// SIMATIC STEP 7 (V5.x) project EuroAsiaFood_V00_00_01
// station: Hardware
// station: SIMATIC 300(1)
// station: P_ADR_BUS
// station: Hardware
// station: SIMATIC 300(1)
// station: P_ADR_BUS

SYMBOL_TABLE
"CMs_SIMULATION_DB"	DB 2	FB 2	// Simulation
"DB3 CPU Daten"	DB 3	DB 3	// Globaldaten
"DB4 Motordaten für FUs"	DB 4	DB 4	// Motordaten für Frequenzumformer
"DB30 Daten von/an FG"	DB 30	FB 30
"DB32 Inputs"	DB 32	FB 32
"DB33 Outputs"	DB 33	FB 33
"DB34 Faults"	DB 34	FB 34
"DB35 Acknolegments"	DB 35	DB 35	// Quittierungen
"DB92 Eingänge AVP"	DB 92	FB 92
"CMs_MOTOR_1Q1I_DB"	DB 901	FB 901	// Motor 1QII
"LINE1"	DB 1000	FB 1000	// Line FB
"CONTAINERSTATION CST01"	DB 1001	FB 1001
"RECEIVER REC01"	DB 1011	FB 1011
"REC01"	DB 1012	FB 1011
"VP01"	DB 1051	FB 1051
"VACUUM PUMP VP01_02 SF01"	DB 1081	FB 1081
"RecipeData"	DB 1111	DB 1111	// Recipes
"test"	DB 2222	DB 2222
"FREQUENCY CONVERTERS"	DB 4900	FB 4900
"FC VACUUM PUMP"	DB 10001	FB 4901	// Vacuum Pump FC
"FC ROTARY FEEDER REC01"	DB 10002	FB 4901	// Rotary Feeder REC01 FC
"CMs_SIMULATION"	FB 2	FB 2	// Simulation
"FB4 Frequenzumformer"	FB 4	FB 4	// Frequenzumformer
"FB30 Daten von/an  FG"	FB 30	FB 30	// Daten von / an Farbgrafik
"FB31 Mode Objekte an FG"	FB 31	FB 31	// Mode der Objekte an Farbgrafik
"FB32 Eingaege an FG"	FB 32	FB 32	// Eingänge der an Farbgrafik
"FB33 Ausgaege an FG"	FB 33	FB 33	// Ausgänge der an Farbgrafik
"FB34 Störbearbeitung"	FB 34	FB 34	// Faults
"FB92 Eingänge AVP"	FB 92	FB 92	// reserve
"CMs_MOTOR_1Q1I"	FB 901	FB 901	// Motor 1QII
"****PRODUCTION****"	FB 1000	FB 1000	// Call Line FBs
"CONTAINERSTATION"	FB 1001	FB 1001	// HP01 and HP02
"RECEIVER"	FB 1011	FB 1011	// Receiver REC01
"VACUUM PUMP"	FB 1051	FB 1051
"VACUUMPUMP"	FB 1081	FB 1081	// BLOWER FB
"*** FCs ***"	FB 4900	FB 4900	// Frequency Converters
"FREQ.CONVERTER"	FB 4901	FB 4901	// Frequency Convertors Calls
"FU SEW DFE32B - PN_REL"	FB 6119	FB 6119
"FU SEW DFE32B - PN"	FB 60119	FB 60119	// SEW Profinet
"FC2 Taktgeber_Timernachb"	FC 2	FC 2	// Taktgeber mit Timernachbildung
"FC3 Timernachbildung"	FC 3	FC 3	// Timernachbildung SA,SE,SV,SI
"FC4 Blocktransfer ANY-Q"	FC 4	FC 4	// Block transferieren mit ANY-Zeiger als Quelle
"FC5 Blocktransfer"	FC 5	FC 5	// Block transferieren, Datenwort schreiben
"FC6 Datenbit zuw./abfr."	FC 6	FC 6	// Datenbit zuweisen oder abfragen
"FC7 Tabelle auslesen"	FC 7	FC 7	// Tabelle auslesen
"FC8 ANY-Zeiger zerlegen"	FC 8	FC 8	// ANY-Zeiger in DB,DW,Länge zerlegen
"FC10 Analogwert r/w"	FC 10	FC 10	// Analogwert lesen/schreiben
"FC13 Standardsignale"	FC 13	FC 13	// Standardsignale
"FC16 Störauswertung"	FC 16	FC 16	// Störauswertung
"FC20 Motor 1A1E"	FC 20	FC 20	// Motor Objekt 1 (1 Ausgang, 1 Eingang)
"FC21 Ventil 1A0-2E"	FC 21	FC 21	// Ventil Objekt 1 (1 Ausgang, 0-2 Eingänge)
"FC22 Ventil 2A2E"	FC 22	FC 22	// Ventil Objekt 2 (2 Ausgänge, 2Eingänge)
"FC23 Ventil 1-10A"	FC 23	FC 23	// Ventil Objekt 3 (Ansteuerung von max. 10 getakteten Ventilen)
"FC24 Binär-E"	FC 24	FC 24	// Binär-Eingangs Objekt
"FC25 Lamp"	FC 25	FC 25
"AnalogueIn"	FC 28	FC 28
"PressureAi"	FC 29	FC 29	// FU Objekt
"FC30 DB vorbelegen"	FC 30	FC 30	// Datenbaustein vorbelegen
"FC40 copy Obj-SST Master"	FC 40	FC 40	// Objekt-Schnittstelle kopieren Master
"FC41 copy Obj-SST Slave"	FC 41	FC 41	// Objekt-Schnittstelle kopieren Slave
"FC47 Tabelle schreiben"	FC 47	FC 47	// Eintrag in Tabelle schreiben
"FC104 Blocktransf. ANY-Z"	FC 104	FC 104
"FC113 Standardsignale 2"	FC 113	FC 113	// Standardsignale
"FC6079 SimAnalog"	FC 6079	FC 6079	// simulate analog signal using sin()
"FC6091 SimValve3A3E"	FC 6091	FC 6091	// simulate valve 3A3E (sealed hose diverter)
"FC6092 SimValveDOS"	FC 6092	FC 6092	// simulate valve 2A2E (dosing valve)
"FC6093 SimValveDS"	FC 6093	FC 6093	// simulate valve 2A2E (double seat)
"FC6094 SimMotor2A2E"	FC 6094	FC 6094	// simulate motor 2A2E
"FC6095 SimValve2A2E"	FC 6095	FC 6095	// simulate valve 2A2E
"FC6096 SimValve1AE1"	FC 6096	FC 6096	// simulate valve 1AE1
"FC6097 SimValve1A1E"	FC 6097	FC 6097	// simulate valve 1A1E
"FC6098 SimValve1A2E"	FC 6098	FC 6098	// simulate valve 1A2E
"FC6099 SimMotor1A1E"	FC 6099	FC 6099	// simulate motor 1A1E
"I 4.0"	I 4.0	BOOL
"02_01_101_Gn"	I 4.1	BOOL	// Production area PMP01 valve fresh air valve
"I 4.2"	I 4.2	BOOL
"02_02_101_Gp"	I 4.3	BOOL	// Production area REC01 valve angle valve
"I 4.4"	I 4.4	BOOL
"I 4.5"	I 4.5	BOOL
"I 4.6"	I 4.6	BOOL
"01_01_101_Gp"	I 4.7	BOOL	// Material preparation CST01 valve fresh air valve
"I 5.0"	I 5.0	BOOL
"02_01_101_Gp"	I 5.1	BOOL	// Production area PMP01 valve fresh air valve
"I 5.2"	I 5.2	BOOL
"02_02_101_Gn"	I 5.3	BOOL	// Production area REC01 valve angle valve
"I 5.4"	I 5.4	BOOL
"I 5.5"	I 5.5	BOOL
"I 5.6"	I 5.6	BOOL
"01_01_101_Gn"	I 5.7	BOOL	// Material preparation CST01 valve fresh air valve
"02_02_601_Lp"	I 6.0	BOOL	// Production area REC01 input high level indicator
"02_02_602_Gn"	I 6.1	BOOL	// Production area REC01 input pendulum flap
"I 6.2"	I 6.2	BOOL
"I 6.3"	I 6.3	BOOL
"I 6.4"	I 6.4	BOOL
"I 6.5"	I 6.5	BOOL
"I 6.6"	I 6.6	BOOL
"10_01_601_ES"	I 6.7	BOOL	// System System input fault fuse
"01_01_601_H"	I 10.0	BOOL	// Material preparation CST01 input illuminated push button
"01_01_602_H"	I 10.1	BOOL	// Material preparation CST01 input illuminated push button
"01_01_603_H"	I 10.2	BOOL	// Material preparation CST01 input push button
"I 10.3"	I 10.3	BOOL
"02_03_601_ES"	I 10.4	BOOL	// Production area PAK01 input PFC
"02_03_602_ES"	I 10.5	BOOL	// Production area PAK01 input PFC
"I 10.6"	I 10.6	BOOL
"I 10.7"	I 10.7	BOOL
"I 11.0"	I 11.0	BOOL
"I 11.1"	I 11.1	BOOL
"I 11.2"	I 11.2	BOOL
"I 11.3"	I 11.3	BOOL
"I 11.4"	I 11.4	BOOL
"I 11.5"	I 11.5	BOOL
"I 11.6"	I 11.6	BOOL
"I 11.7"	I 11.7	BOOL
"M0.0 LockManualMode"	M 0.0	BOOL	// central lock for manual mode
"M0.1 Constant1"	M 0.1	BOOL	// flag constant 1
"M0.2 Constant0"	M 0.2	BOOL	// flag constant 0
"M0.3 Reset"	M 0.3	BOOL	// general reset
"M0.4 CotrolVoltageOn"	M 0.4	BOOL	// control voltage on
"M0.5 SimulationInternal"	M 0.5	BOOL	// simulation internal on
"M0.6 SimulationAVP"	M 0.6	BOOL	// simulation with AVP
"M0.7 BatteryEmpty"	M 0.7	BOOL	// battery empty
"M1.0 AcknowledgeFault"	M 1.0	BOOL	// acknowledge fault (general)
"M1.1 Fault(General)"	M 1.1	BOOL	// fault (general)
"M1.2 NewFault(General)"	M 1.2	BOOL	// new fault (first indication)
"M1.3 CompleteRestart"	M 1.3	BOOL	// complete restart PLC
"M1.4 RestartPLC"	M 1.4	BOOL	// restart PLC
"M1.5 Lamp Test"	M 1.5	BOOL	// Lamp Test
"M1.6 ClockLevelIndicato"	M 1.6	BOOL	// clock for debouncing level indicators
"M1.7 ClockTimerFunction"	M 1.7	BOOL	// clock for timer-FCs
"M2.0 Flag0,1Sec"	M 2.0	BOOL	// flag clock 0,1 sec
"M2.1 Flag0,2Sec"	M 2.1	BOOL	// flag clock 0,2 sec
"M2.2 Flag0,4Sec"	M 2.2	BOOL	// flag clock 0,4 sec
"M2.3 Flag0,5Sec"	M 2.3	BOOL	// flag clock 0,5 sec
"M2.4 Flag0,8Sec"	M 2.4	BOOL	// flag clock 0,8 sec
"M2.5 Flag1,0Sec"	M 2.5	BOOL	// flag clock 1,0 sec
"M2.6 Flag1,6Sec"	M 2.6	BOOL	// flag clock 1,6 sec
"M2.7 Flag2,0Sec"	M 2.7	BOOL	// flag clock 2,0 sec
"M3.0 EdgeClock0,1Sec"	M 3.0	BOOL	// flank flag clock 0,1 sec
"M3.1 EdgeClock0,2Sec"	M 3.1	BOOL	// flank flag clock 0,2 sec
"M3.2 EdgeClock0,4Sec"	M 3.2	BOOL	// flank flag clock 0,4 sec
"M3.3 EdgeClock0,5Sec"	M 3.3	BOOL	// flank flag clock 0,5 sec
"M3.4 EdgeClock0,8Sec"	M 3.4	BOOL	// flank flag clock 0,8 sec
"M3.5 EdgeClock1,0Sec"	M 3.5	BOOL	// flank flag clock 1,0 sec
"M3.6 EdgeClock1,6Sec"	M 3.6	BOOL	// flank flag clock 1,6 sec
"M3.7 EdgeClock2,0Sec"	M 3.7	BOOL	// flank flag clock 2,0 sec
"M4.0 ImpulseClock0,1Sec"	M 4.0	BOOL	// impulse flag clock 0,1 sec
"M4.1 ImpulseClock0,2Sec"	M 4.1	BOOL	// impulse flag clock 0,2 sec
"M4.2 ImpulseClock0,4Sec"	M 4.2	BOOL	// impulse flag clock 0,4 sec
"M4.3 ImpulseClock0,5Sec"	M 4.3	BOOL	// impulse flag clock 0,5 sec
"M4.4 ImpulseClock0,8Sec"	M 4.4	BOOL	// impulse flag clock 0,8 sec
"M4.5 ImpulseClock1,0Sec"	M 4.5	BOOL	// impulse flag clock 1,0 sec
"M4.6 ImpulseClock1,6Sec"	M 4.6	BOOL	// impulse flag clock 1,6 sec
"M4.7 ImpulseClock2,0Sec"	M 4.7	BOOL	// impulse flag clock 2,0 sec
"Service Mode ExpertMode"	M 9.5	BOOL	// Service Mode Expert
"GlobalLampTesting"	M 9.7	BOOL	// Lamp Test
"Release Man Mode Motors"	M 10.0	BOOL	// Man Mode for Motors is released
"AckObligatoryMotors"	M 10.1	BOOL	// Faults for Motors needs to Ack
"Release Man Mode Valves"	M 11.0	BOOL	// Man Mode for Valves is released
"AckObligatoryValves"	M 11.1	BOOL	// Faults for Valves needs to Ack
"M37.0 AckObligationMotor"	M 37.0	BOOL	// acknowledging motor faults obligatory
"M37.1 AckObligationValve"	M 37.1	BOOL	// acknowledging valve faults obligatory
"M37.2 AckObligationOther"	M 37.2	BOOL	// acknowledging other faults obligatory
"M37.3 AckObligationISO"	M 37.3	BOOL	// acknowledging motor isolator faults obligatory
"M37.4 AckObligationSecSw"	M 37.4	BOOL	// acknowledging safety switch faults obligatory
"M37.5 AckObligationMotBr"	M 37.5	BOOL	// acknowledging motor breaker faults obligatory
"M37.6 AckObligation = 1"	M 37.6	BOOL	// general acknowledging obligatory
"M37.7 AckObligation = 0"	M 37.7	BOOL	// no acknowledging obligatory
"MW 6 Timer Val Cycle FCs"	MW 6	INT	// Zeitwert Takt-FCs in 0,1s
"OB 1 Zyklisches Prg."	OB 1	OB 1	// Zyklisches Programm
"OB 80 Zeitfehler-OB"	OB 80	OB 80	// Zeitfehler-OB
"OB 82 Diagnosealarm-OB"	OB 82	OB 82	// Diagnosealamrn-OB
"OB 83 Ziehen-/Stecken-OB"	OB 83	OB 83	// Ziehen-/Stecke-OB
"OB 85 Prgablauffehler-OB"	OB 85	OB 85	// Programmablauffehler-OB
"OB 86 Baugr träger-OB"	OB 86	OB 86	// Baugruppenträgerausfall-OB
"OB 87 Kommunikations-OB"	OB 87	OB 87	// Kommunikationsfehler-OB
"OB 100 Neustart-OB"	OB 100	OB 100	// Neustart-OB
"OB 121 Programmierf-OB"	OB 121	OB 121	// Programmierfehler-OB
"02_01_401_PI"	PIW 200	WORD	// Production area PMP01 analog signal pressure transmitter
"PIW 202"	PIW 202	WORD
"PIW 204"	PIW 204	WORD
"PIW 206"	PIW 206	WORD
"PQW 200"	PQW 200	WORD
"PQW 202"	PQW 202	WORD
"Q 4.0"	Q 4.0	BOOL
"02_01_101_UVn"	Q 4.1	BOOL	// Production area PMP01 valve fresh air valve
"Q 4.2"	Q 4.2	BOOL
"02_02_101_UVp"	Q 4.3	BOOL	// Production area REC01 valve angle valve
"02_02_102_UVp"	Q 4.4	BOOL	// Production area REC01 valve filter cleaning
"02_02_103_UVp"	Q 4.5	BOOL	// Production area REC01 valve rapper
"Q 4.6"	Q 4.6	BOOL
"01_01_101_UVp"	Q 4.7	BOOL	// Material preparation CST01 valve fresh air valve
"Q 5.0"	Q 5.0	BOOL
"Q 5.1"	Q 5.1	BOOL
"Q 5.2"	Q 5.2	BOOL
"Q 5.3"	Q 5.3	BOOL
"Q 5.4"	Q 5.4	BOOL
"Q 5.5"	Q 5.5	BOOL
"Q 5.6"	Q 5.6	BOOL
"Q 5.7"	Q 5.7	BOOL
"01_01_501_H"	Q 10.0	BOOL	// Material preparation CST01 output illuminated push button
"01_01_502_H"	Q 10.1	BOOL	// Material preparation CST01 output illuminated push button
"Q 10.2"	Q 10.2	BOOL
"Q 10.3"	Q 10.3	BOOL
"01_02_501_ES"	Q 10.4	BOOL	// Material preparation MI01 output PFC
"Q 10.5"	Q 10.5	BOOL
"Q 10.6"	Q 10.6	BOOL
"Q 10.7"	Q 10.7	BOOL
"Q 11.0"	Q 11.0	BOOL
"Q 11.1"	Q 11.1	BOOL
"Q 11.2"	Q 11.2	BOOL
"Q 11.3"	Q 11.3	BOOL
"Q 11.4"	Q 11.4	BOOL
"10_01_501_H"	Q 11.5	BOOL	// System System output pilot lamp
"10_01_502_H"	Q 11.6	BOOL	// System System output pilot lamp
"10_01_503_H"	Q 11.7	BOOL	// System System output pilot lamp
"SET_CLK"	SFC 0	SFC 0	// Set System Clock
"READ_CLK"	SFC 1	SFC 1	// Read System Clock
"DPRD_DAT"	SFC 14	SFC 14	// Read Consistent Data of a Standard DP Slave
"DPWR_DAT"	SFC 15	SFC 15	// Write Consistent Data to a Standard DP Slave
"BLKMOV"	SFC 20	SFC 20	// Copy Variables
"TEST_DB"	SFC 24	SFC 24	// Test Data Block
"RDSYSST"	SFC 51	SFC 51	// Read a System Status List or Partial List
"TIME_TCK"	SFC 64	SFC 64	// Read the System Time
"Schnittstelle FU"	UDT 1	UDT 1
"Cmod_AnalogueIn"	UDT 128	UDT 128
"Cmod_PressureAi"	UDT 129	UDT 129
"VAT_1"	VAT 1	
END_SYMBOL_TABLE

TYPE "Schnittstelle FU"	// UDT 1
VERSION : 0.1
  STRUCT
   Schnittstelle_FU : STRUCT
    von : STRUCT
     Istfrequenz : REAL ;
     reserve : ARRAY  [4 .. 17 ] OF BYTE ;
     Statusbits : STRUCT
      Bereit : BOOL ;
      Laeuft : BOOL ;
      Stoerung : BOOL ;
     END_STRUCT ;
    END_STRUCT ;
    an : STRUCT
     Antwort_DB : INT ;
     Antwort_DW : INT ;
     Sollfrequenz : REAL ;
     Motordatensatz_Nummer : INT ;
     reserve : ARRAY  [10 .. 17 ] OF BYTE ;
     Steuerbits : STRUCT
      Anforderung : BOOL ;
      Freigabe : BOOL ;
      Linkslauf : BOOL ;
     END_STRUCT ;
    END_STRUCT ;
   END_STRUCT ;
  END_STRUCT ;	
END_TYPE

TYPE "Cmod_AnalogueIn"	// UDT 128
VERSION : 0.1
  STRUCT
   parameter : STRUCT
    AnalogInOn : BOOL ;	//Activate popup
    reserve1 : BOOL ;
    reserve2 : BOOL ;
    switching_number_counter : BOOL ;	//Counter for operating cycles
    switch_level : BOOL ;	//view/edit switch level
    switch_hysteresis : BOOL ;	//view/edit switch hysteresis
    reserve_6 : BOOL ;
    reserve_7 : BOOL ;
    alarm_high : BOOL ;	//view/edit alarm high
    alarm_low : BOOL ;	//view/edit alarm low
    alarm_hyst : BOOL ;	//view/edit alarm hysteresis
    reserve_11 : BOOL ;
    reserve_12 : BOOL ;
    reserve_13 : BOOL ;
    reserve_14 : BOOL ;
    reserve_15 : BOOL ;
    uom_code : INT ;	//code for unit of measurement
   END_STRUCT ;
   ManModeAct : BOOL ;	//0=Automode; 1=Manualmode
   ManModeOp : BOOL ;	//0=Automode; 1=Manualmode
   ManModeLock : BOOL ;	//Lock manual mode
   SystemOn : BOOL ;
   ScalingErr : BOOL ;
   OVErr : BOOL ;
   AlarmHi : BOOL ;	//Alarm high
   AlarmHiEn : BOOL ;	//Alarm high enable
   AlarmHiAck : BOOL ;	//Alarm high acknowledge
   AlarmLo : BOOL ;	//Alarm low
   AlarmLoEn : BOOL ;	//Alarm low enable
   AlarmLoAck : BOOL ;	//Alarm low acknowledge
   Switch : BOOL ;
   SwitchEn : BOOL ;
   PVAct : REAL ;
   ManModePV : REAL ;	//Value for manual mode
   AlarmHiPV : REAL ;
   AlarmLoPV : REAL ;
   AlarmHystPV : REAL ;
   SwitchLevelPV : REAL ;
   SwitchHystPV : REAL ;
   cyclecounter : STRUCT
    Reset : BOOL ;	//Reset operating cycle counter
    Warning : BOOL ;	//Warning time 1 elapsed
    Alarm : BOOL ;	//Alarm time 2 elapsed
    Edge : BOOL ;	//Intern used flag
    CountAct : REAL ;	//Actual number of cycles (cycle counter)
    CountWarning : REAL ;	//Set value for generate the warning
    CountAlarm : REAL ;	//Set value for generate the alarm
   END_STRUCT ;
   object_state : INT ;
  END_STRUCT ;	
END_TYPE

TYPE "Cmod_PressureAi"	// UDT 129
AUTHOR : gea
VERSION : 1.0
  STRUCT
   parameter : STRUCT
    PressureAIOn : BOOL  := TRUE;	//Activate popup
    reserve1 : BOOL ;
    reserve2 : BOOL ;
    counterOverPressure : BOOL  := TRUE;	//Counter for operating cycles
    counterEmptyPressure : BOOL ;	//Counter for operating cycles
    counterActivePressure : BOOL ;	//Counter for operating cycles
    reserve_6 : BOOL ;
    reserve_7 : BOOL ;
    OverPressure : BOOL  := TRUE;	//view/edit OverPressure levels
    EmptyPressure : BOOL  := TRUE;	//view/edit EmptyPressure levels
    ActivePressure : BOOL  := TRUE;	//view/edit ActivePressure levels
    reserve_13 : BOOL ;
    ManOpSimEn : BOOL  := TRUE;
    MapOpAdjustEn : BOOL  := TRUE;
    reserve_14 : BOOL ;
    reserve_15 : BOOL ;
    uom_code : INT ;	//code for unit of measurement
   END_STRUCT ;
   ManModeAct : BOOL ;	//0=Automode; 1=Manualmode
   ManModeOp : BOOL ;	//0=Automode; 1=Manualmode
   ManModeLock : BOOL ;	//Lock manual mode
   ManOpPressureEmpty : BOOL ;
   ManOpPressureConveying : BOOL ;
   ManOpPressureAlarm : BOOL ;
   ManOpPressureAdjust : BOOL ;
   SystemOn : BOOL ;
   ScalingErr : BOOL ;
   OVErr : BOOL ;
   ParErr : BOOL ;
   fOverpressure : BOOL ;
   fOverpressureEn : BOOL ;
   fOverpressureAck : BOOL ;
   Overpressure : BOOL ;
   Emptypressure : BOOL ;
   ActivePressure : BOOL ;
   Active : BOOL  := TRUE;
   AdjustRelease : BOOL ;
   AdjustPulse : BOOL  := TRUE;
   ManAdjustReq : BOOL ;
   ManAdjustRdy : BOOL  := TRUE;
   CounterReset : BOOL ;	//Reset operating cycle counter
   CounterEdge : BOOL ;	//Intern used flag
   PVAct : REAL ;
   PressureOffset : REAL ;
   MaxOverpressurePV : REAL ;
   MinOverpressurePV : REAL ;
   EmptypressurePV : REAL ;
   ActivePressurePV : REAL ;
   EmptyDelay : INT  := 5;
   ActiveDelay : INT  := 5;
   AlarmDelay : INT  := 10;
   EmptyDelayCounter : INT ;
   ActiveDelayCounter : INT ;
   AlarmDelayCounter : INT ;
   CounterAct : REAL ;	//Actual number of cycles (cycle counter)
   object_state : INT ;
  END_STRUCT ;	
END_TYPE

FUNCTION_BLOCK "CMs_SIMULATION"	// FB 2
TITLE = Simulation
//Creation:
//Date:            Author:                                               Version
//--------------------------------------------------------------------------------
//20.09.2019      Ilia                                                   01.00.00
//
//Changes:
//No. Date:        Who       Description                           Mark   Version 
//--------------------------------------------------------------------------------
//01
//________________________________________________________________________________
//Function:
//
VERSION : 0.1
VAR
  REC01 : STRUCT
   Weight : REAL ;
   SpeedFilling : REAL ;
   SpeedDischarging : REAL ;
  END_STRUCT ;
  HP03 : STRUCT
   Weight : REAL ;
   SpeedFilling : REAL ;
   SpeedDischarging : REAL ;
  END_STRUCT ;
END_VAR
BEGIN
NETWORK
TITLE = simulation condition
      AN    "M0.5 SimulationInternal";
      BEC;
NETWORK
TITLE = ----------------------------PMP01-----------------------------
NETWORK
TITLE = Rotary Valve - direct FC
      A     "M0.1 Constant1";
      =     "10_01_601_ES";
NETWORK
TITLE = Fresh Air Valve 1Q2I PMP01
      CALL  "FC6098 SimValve1A2E" (
           o_ValveOn                := "02_01_101_UVn",
           i_ValveOn                := "02_01_101_Gn",
           i_ValveOff               := "02_01_101_Gp");
NETWORK
TITLE = ----------------------------REC01-----------------------------
NETWORK
TITLE = Fresh Air Valve 1Q2I REC01
      CALL  "FC6098 SimValve1A2E" (
           o_ValveOn                := "02_02_101_UVp",
           i_ValveOn                := "02_02_101_Gp",
           i_ValveOff               := "02_02_101_Gn");
NETWORK
TITLE = Filter Cleaning Valve 1Q0I
NETWORK
TITLE = -----------------------CST01------------------------------------
NETWORK
TITLE = Fresh Air Valve 1Q2I CST01
      CALL  "FC6098 SimValve1A2E" (
           o_ValveOn                := "01_01_101_UVp",
           i_ValveOn                := "01_01_101_Gp",
           i_ValveOff               := "01_01_101_Gn");
NETWORK
TITLE =
NETWORK
TITLE = ------------------------VACUUM PUMP-----------------------------
NETWORK
TITLE = VP01
// Direct FC
      A     "M0.1 Constant1";
      =     "02_02_602_Gn";
NETWORK
TITLE = VP02
      CALL  "FC6099 SimMotor1A1E" (
           o_MotorOn                := "Q 4.0",
           Isolators                := TRUE,
           i_MotorOn                := "I 4.0",
           i_IsoMotor               := "02_02_601_Lp");
NETWORK
TITLE = PFKs HP
      A     "M0.1 Constant1";
      =     I 9.4;
NETWORK
TITLE = NH is OK
      A     "M0.1 Constant1";
      =     "I 5.2";
      =     "01_01_101_Gn";
END_FUNCTION_BLOCK

FUNCTION_BLOCK "FB4 Frequenzumformer"	// FB 4
TITLE = Steuerung von SEW-Frequenzumf. mit DFP21B über Profibus-DP
//Building:
//Date         Editor                                                     Version
//--------------------------------------------------------------------------------
//11.12.06     R.Schaffert (sra)                                          01.00.00
//
//Modifications:
//No. Date     Edit  Description                                    Index Version
//--------------------------------------------------------------------------------
//01  12.04.07 sra   Ausgangsstrom in Ampere ausgeben               (001) 01.00.01
//02  23.06.10 sra   Betriebsmeldung mit Komm.fehlern erweitert     (002) 01.00.02
//03  19.10.11 sra   Begrenzung maximale Solldrehzahl               (003) 01.01.00
//04  19.03.12 sra   Änderung wegen Firmwareänderung SEW            (004) 01.01.01
//05  23.07.14 sra   Umschaltung Parametersatz eingefügt            (005) 01.02.00
//05  23.09.14 sra   Fehlerbeseitigung "Warnung"                    (006) 01.02.01
//06  23.11.15 kst   Fehlerbeseitigung allgemein                    (007) 01.03.00
//07  17.02.16 sra   out_FB_Fehlermeldung = INT                     (008) 01.03.01
//________________________________________________________________________________
//Functional description:
//
//The block communicates with SEW frequency converters MOVITRAC B via 
//Profibus interface DFP21B.
//
//Note:
//With this frequency converter it is not possible to transfer motor data.
//To be sure that the output value of the current is correct, the paramter 
//nominal motor current at the frequency convetrer must be set to correct value.
//
//Hardware configuration:
//
//Install GSD file in hardware catalogue:
// SEW_6009.GSD (Internet: www.SEW-EURODRIVE.de)
//
//The "Gateway DFP/DFS" Profibus module is then in the hardware catalogue under 
//the menu: "other field devices->Drives->SEW->DPV1->"
//Add this module to hardware and configure following modules
//     Slot 1: Empty
//     Slot 2: Parameter channel (8 byte)  with I/O address Z
//from Slot 3: AS Y Drives (Y x 3PD)       with I/O address Z+8 and following
//             where Y = Number of FCs 
//
//
//!!! The nominal motor frequency, motor speed and the nominal motor current must 
//    be transferred to ensure the block functions correctly.
//
//Settings at DFP21B:
//
//1. Set Profibus address via DIP switches on DFP21B: 
//
//2. Execute auto setup at DFP21B by setting DIP switch 8 (AS) to ON
//   All FCs must be switched on and the SBus address set
//   With the auto setup function (DIP switch "AS") it is possible to set up 
//   DFP21B as the gateway without a PC. The function is executed once when the 
//   DIP switch is switched on. The DIP switch must then remain on. The function 
//   can be executed again by switching the DIP switch off and on again.
//
//
//Frequency converter settings
//
//1. P100 Set setpoint source to SBUS -> value = 10
//
//2. P101 Set control source to SBus -> value 3
//
//3. P301 Set minimum speed in rpm (master value = 15)
//
//4. P302 Set maximum speed in rpm (factory setting = 1500)
//
//5. P303 Set current limit (in % of FC nominal current)
//   (Factory setting =150%)
//
//6. P320 Set automatic motor matching to on (standard setting)
//   (to gauge the motor at start)
//
//7. P500 Switch on speed monitoring
//   (in the case of fault messages P501 increase speed monitoring delay time)
//
//8. P601, P603 and P608 Set binary inputs to ""no function" (=0)
//   Set P602 to 1 = enable (factory setting) DI03 must be bypassed
//
//9. P604 for operation with PTC resistor set to 26 (TF message) otherwise
//.... zeroing.
//   
//11. P881 Set SBus address of respective frequency converter (from 1 in
//    ascending order)
//
//12. P883 Bus monitoring time -> 5 [s]
//
//13. P884 Check SBus baud rate -> value 500/500 kBaud
//
//14. P870-P872 Setpoint description PA1-PA3
//       P870 = control word 1
//       P871 = speed
//       P872 = reserve
//    P873-P876 Actual value description PE1-PE3
//       P873 = status word 1
//       P874 = speed
//       P875 = output current in % of nominal current
//
//Notice to Index/Modification (004):
//The firmware has been changed because some faults must be resetet with an 
//internal function and some other with an acknowledge function. If there has 
//been 
//an fault of the Thermocontact is wasn't necessary to reset the fault and the 
//frequency converter still signals "ready for operation". This also happened 
//with other fault messages. For the Profibus communication it wasn't possible to 
//detect what happend with the motor. Finally the function always signals always 
//a fault message.
//
AUTHOR : sra
FAMILY : AZO
VERSION : 0.0
VAR_INPUT
  in_PEA_Adresse : INT ;	//Basisadresse für EA-Daten im PEA-Bereich
  in_FU_Nummer : INT ;	//FU Nummer zur Berechnung des Offsets der Peripherie-EAs
  in_Auswahl_Param_satz_2 : BOOL ;	//Motorparametersatz 2 wird ausgewählt (bei Ansteuerung von 2 versch. Motortypen)
  in_Freigabe : BOOL ;	//Steuersignal 1 setzen zum Starten des FUs
  in_Linkslauf : BOOL ;	//Frequenzumformer Linkslauf ein
  in_Quittierung_Stoerung : BOOL ;	//Störung quittieren
  in_Sollfrequenz : REAL ;	//Sollfrequenz in Hz
  in_Motorleistungsfaktor : REAL ;	//nicht vorhanden => 0
  in_Motornennfrequenz : REAL ;	//Wertebereich: 0 - 100 Hz
  in_Motornenndrehzahl : REAL ;	//Wertebereich: 0 - 10000 U/min
  in_Motornennstrom : REAL ;	//Wertebereich: 0- ... A !! Hier muss der Stromwert des FUs eingegeben werden !!
  in_Motornennspannung : REAL ;	//nicht vorhanden => 0
  in_Motornennleistung : REAL ;	//nicht vorhanden => 0
END_VAR
VAR_OUTPUT
  out_Istfrequenz : REAL ;	//Istfrequenz in Hz
  out_Istdrehzahl : REAL ;	//Istdrehzahl in U/min
  out_Leistung : REAL ;	//nicht vorhanden => 0
  out_Drehmoment : REAL ;	//nicht vorhanden => 0
  out_Motorspannung : REAL ;	//nicht vorhanden => 0
  out_Ausgangsstrom : REAL ;	//Ausgangsstrom des FU
  out_Stoerung : BOOL ;	//1=Gerätestörung
  out_Warnung : BOOL ;	//1=max. Solldrehzahl überschritten
  out_Sollwert_erreicht : BOOL ;	//zeigt 1 an, wenn Istwert gleich Sollwert ist
  out_laeuft : BOOL ;	//=1 wenn Istdrehzahl > 0
  out_FB_Fehlermeldung : INT ;	//0 = ok ; sonst Fehler_Code_L2Dp (008)
  out_Stoerungsnummer : DINT ;	//Stoerungsnummer, bzw. Betriebszustand wenn keine Störung aktiv
END_VAR
VAR
  reserve : ARRAY  [58 .. 99 ] OF BYTE ;
  Parameterkanal_in : STRUCT
   Verwaltung_Subindex : STRUCT
    Dienst_Kennung_0 : BOOL ;
    Dienst_Kennung_1 : BOOL ;
    Dienst_Kennung_2 : BOOL ;
    Dienst_Kennung_3 : BOOL ;
    Datenlaenge_0 : BOOL ;
    Datenlaenge_1 : BOOL ;
    Handshake : BOOL ;
    Status_Bit : BOOL ;
    Subindex : BYTE ;
   END_STRUCT ;
   Parameter_Index : WORD ;
   Daten_1_2 : INT ;
   Daten_3_4 : INT ;
  END_STRUCT ;
  Parameterkanal_out : STRUCT
   Verwaltung_Subindex : STRUCT
    Dienst_Kennung_0 : BOOL ;
    Dienst_Kennung_1 : BOOL ;
    Dienst_Kennung_2 : BOOL ;
    Dienst_Kennung_3 : BOOL ;
    Datenlaenge_0 : BOOL ;
    Datenlaenge_1 : BOOL ;
    Handshake : BOOL ;
    Status_Bit : BOOL ;
    Subindex : BYTE ;
   END_STRUCT ;
   Parameter_Index : WORD ;
   Daten_1_2 : INT ;
   Daten_3_4 : INT ;
  END_STRUCT ;
  Prozessdatenkanal_in : STRUCT 	//Prozesseingangsdaten
   PI1_Statuswort : STRUCT
    Zustand_Fehlercode : BYTE ;
    Endstufe_freigegeben : BOOL ;
    Umrichter_betriebsbereit : BOOL ;
    PA_Daten_freigegeben : BOOL ;
    reserve_3 : BOOL ;
    akt_Parametersatz_2 : BOOL ;	//0 = 1. Satz; 1 = 2. Satz
    Stoerung_Warnung : BOOL ;
    reserve_6 : BOOL ;	//
    reserve_7 : BOOL ;	//
   END_STRUCT ;
   PI2_Istdrehzahl : INT ;
   PI3_Ausgangsstrom : INT ;
  END_STRUCT ;
  Prozessdatenkanal_out : STRUCT 	//Prozessausgangsdaten
   PO1_Steuerwort : STRUCT
    Drehrichtung : BOOL ;	//0 = rechts; 1 = links
    Motorpoti_auf : BOOL ;	//00=11= keine Änderung; 01=Hochlauf, 02=Tieflauf
    Motorpoti_ab : BOOL ;
    Festsollwerte_0 : BOOL ;	//00 = Feldbus
    Festsollwerte_1 : BOOL ;
    Festsollwert_Umschaltung : BOOL ;
    reserve_14 : BOOL ;
    reserve_15 : BOOL ;
    Reglersperre : BOOL ;	//Freigabe = '110', sonst Halt
    Freigabe_Schnellstop : BOOL ;
    Freigabe_Normalhalt : BOOL ;
    reserve_3 : BOOL ;
    Integratorauswahl : BOOL ;	//0 = Integrator 2; 1 = Integrator 1 (005) noch nicht verwendet
    Parametersatz_2 : BOOL ;	//0 = Parametersatz 1; 1 = Parametersatz 2 (005)
    Reset_Stoerung : BOOL ;	//
    reserve_7 : BOOL ;
   END_STRUCT ;
   PO2_Solldrehzahl : INT ;	//in %
   PO3_keine_Fkt : INT ;
  END_STRUCT ;
  Datenuebertragung : STRUCT
   Schritt_aktiv : BOOL ;
  END_STRUCT ;
END_VAR
VAR_TEMP
  IO_Adr_Parameterkanal : WORD ;
  IO_Adr_Prozessdatenkanal : WORD ;
  Ret_Val_SFC14_1 : INT ;
  Ret_Val_SFC14_2 : INT ;
  Ret_Val_SFC15_1 : INT ;
  Ret_Val_SFC15_2 : INT ;
  Solldrehzahl_tmp : REAL ;
END_VAR
BEGIN
NETWORK
TITLE = Bausteinende wenn PEA-Adresse = 0
      L     #in_PEA_Adresse;
      L     0;
      ==I;
      BEC;
NETWORK
TITLE = Simulation
//Über die Simulaitonsmerker "M 0.5 Simulation intern" oder "M 0.6 Simulation 
//AVP" 
//wird die Funktion des FUs simuliert:
//- Fehler werden zurückgesetzt
//- Bei Freigabe Istdrehzahl=Solldrehzahl, Betrieb und Solldrehzahl erreicht = 
//True
      O     "M0.5 SimulationInternal";
      O     "M0.6 SimulationAVP";
      JCN   NSIM;
      SET;
      R     #out_Stoerung;
      L     L#0;
      T     #out_Stoerungsnummer;
      A     #in_Freigabe;
      =     #out_laeuft;
      =     #out_Sollwert_erreicht;	// (007)
      L     #in_Sollfrequenz;
      JC    SIMD;
      L     0.000000e+00;
SIMD: T     #out_Istfrequenz;
      BEU;
NSIM: NOP   0;
NETWORK
TITLE = Daten von FU einlesen
//UFP-Parameter und FU-Daten auslesen mit SFC14
//PEA_Adresse zeigt auf den Anfang des EA-Bereiches.
// 8-Byte Parameterkanal
      L     #in_PEA_Adresse;
      T     #IO_Adr_Parameterkanal;
      CALL  "DPRD_DAT" (
           LADDR                    := #IO_Adr_Parameterkanal,
           RET_VAL                  := #Ret_Val_SFC14_1,
           RECORD                   := #Parameterkanal_in);
// 6-Byte Prozessdatenkanal
      L     #in_FU_Nummer;
      +     -1;
      L     6;	// Länge eines Parameterkanals je FU
      *I;
      L     #in_PEA_Adresse;
      +I;
      L     8;	// Offset für Parameterkanal
      +I;
      T     #IO_Adr_Prozessdatenkanal;	// Daten des jeweiligen FU = PEA-Adresse + 8 Byte + (FU-Nr. - 1) * 6
      CALL  "DPRD_DAT" (
           LADDR                    := #IO_Adr_Prozessdatenkanal,
           RET_VAL                  := #Ret_Val_SFC14_2,
           RECORD                   := #Prozessdatenkanal_in);
NETWORK
TITLE = Betriebsmeldung
      A     #Prozessdatenkanal_in.PI1_Statuswort.Endstufe_freigegeben;
      A     #Prozessdatenkanal_in.PI1_Statuswort.Umrichter_betriebsbereit;
      A     #Prozessdatenkanal_in.PI1_Statuswort.PA_Daten_freigegeben;
      A(;	// (002)
      L     #Ret_Val_SFC14_2;	// (002)
      L     0;	// (002)
      ==I;	// (002)
      );	// (002)
      =     #out_laeuft;
NETWORK
TITLE = Sollwert erreicht
      L     #in_Sollfrequenz;
      L     #out_Istfrequenz;
      -R;
      ABS;
      L     1.000000e+00;
      <R;
      =     #out_Sollwert_erreicht;
NETWORK
TITLE = Istdrehzahl auswerten
//Istdrehzahl in 0,2 U/min
      L     #Prozessdatenkanal_in.PI2_Istdrehzahl;
      ITD;
      DTR;
      L     5.000000e+00;
      /R;
      T     #out_Istdrehzahl;
NETWORK
TITLE = Istfrequenz auswerten
//Istfrequenz (in Hz) = Istdrehzahl (in 0,2 U/min) / 5 * Nennfrequenz / 
//Nenndrehzahl 
      L     #Prozessdatenkanal_in.PI2_Istdrehzahl;	// (1 == 0,2 U/min)
      ITD;
      DTR;
      L     5.000000e+00;
      /R;
      L     #in_Motornennfrequenz;
      *R;
      L     #in_Motornenndrehzahl;
      /R;
      T     #out_Istfrequenz;	// in Hz
      L     0.000000e+00;	//  wenn kleiner 0 dann negieren 
      <R;
      JCN   E_IF;
      L     #out_Istfrequenz;
      L     -1.000000e+00;
      *R;
      T     #out_Istfrequenz;
E_IF: NOP   0;
NETWORK
TITLE = Stromwert auswerten
      L     #Prozessdatenkanal_in.PI3_Ausgangsstrom;	// in % des FU-Nennstomes 
      ITD;
      DTR;
      L     1.000000e+02;	// (001)
      /R;	// (001)
      L     #in_Motornennstrom;	// (001)
      *R;	// (001)
      T     #out_Ausgangsstrom;
NETWORK
TITLE = Störungsbit auswerten
//Störungsbit aus Statuswort auswerten
//      UN    #Prozessdatenkanal_in.PI1_Statuswort.Umrichter_betriebsbereit    // (004)
      A     #Prozessdatenkanal_in.PI1_Statuswort.Stoerung_Warnung;
      =     #out_Stoerung;
NETWORK
TITLE = Störung resetten
//Störung resetten
      A     #in_Quittierung_Stoerung;
      A     #Prozessdatenkanal_in.PI1_Statuswort.Stoerung_Warnung;
      =     #Prozessdatenkanal_out.PO1_Steuerwort.Reset_Stoerung;
NETWORK
TITLE = Gerätezustand / Störungsnummer des Frequenzumformers auslesen
//Gerätezustand wenn Bit Störung/Warnung = 0
//Störungsnummer wenn Bit Störung/Warnung = 1
      L     #Prozessdatenkanal_in.PI1_Statuswort.Zustand_Fehlercode;
      ITD;
      T     #out_Stoerungsnummer;
// Störmeldung nur wenn Bit Störung = 1
      A     #Prozessdatenkanal_in.PI1_Statuswort.Stoerung_Warnung;
      JC    ESTO;
      L     0;
      T     #out_Stoerungsnummer;
ESTO: NOP   0;
NETWORK
TITLE = Freigabebefehl bearbeiten
//      CLR   // (006)
      AN    #in_Freigabe;	// (006)
      A     #in_Auswahl_Param_satz_2;	// (006)
      AN    #Prozessdatenkanal_in.PI1_Statuswort.akt_Parametersatz_2;	// (006)
      O;
      AN    #in_Freigabe;	// (006)
      AN    #in_Auswahl_Param_satz_2;	// (006)
      A     #Prozessdatenkanal_in.PI1_Statuswort.akt_Parametersatz_2;	// (006)
      =     #Prozessdatenkanal_out.PO1_Steuerwort.Reglersperre;
      SET;
      =     #Prozessdatenkanal_out.PO1_Steuerwort.Freigabe_Schnellstop;
      A     #in_Freigabe;
      =     #Prozessdatenkanal_out.PO1_Steuerwort.Freigabe_Normalhalt;
NETWORK
TITLE = Parametersatz 2 auswählen
//(005) 
//Über dieses Bit kann der Motorparametersatz 2 des FUs angewählt werden
      A     #in_Auswahl_Param_satz_2;	// (005)
      =     #Prozessdatenkanal_out.PO1_Steuerwort.Parametersatz_2;	// (005)
NETWORK
TITLE = Parametersatz 2 auswählen
//(005) 
//Über dieses Bit kann zwischen Integrator 1 und Integrator 2 umgeschaltet werden
//wird nicht verwendet und dauerhaft auf 0 gesetzt
      CLR;	// (005)
      =     #Prozessdatenkanal_out.PO1_Steuerwort.Integratorauswahl;	// (005)
NETWORK
TITLE = Belegung der restlichen Steuerbits
      CLR;
      =     #Prozessdatenkanal_out.PO1_Steuerwort.reserve_3;
      =     #Prozessdatenkanal_out.PO1_Steuerwort.Integratorauswahl;
//      =     #Prozessdatenkanal_out.PO1_Steuerwort.Parametersatz_2 // (005)
      =     #Prozessdatenkanal_out.PO1_Steuerwort.reserve_7;
      =     #Prozessdatenkanal_out.PO1_Steuerwort.Motorpoti_auf;
      =     #Prozessdatenkanal_out.PO1_Steuerwort.Motorpoti_ab;
      =     #Prozessdatenkanal_out.PO1_Steuerwort.Festsollwerte_0;
      =     #Prozessdatenkanal_out.PO1_Steuerwort.Festsollwerte_1;
      =     #Prozessdatenkanal_out.PO1_Steuerwort.Festsollwert_Umschaltung;
      =     #Prozessdatenkanal_out.PO1_Steuerwort.reserve_14;
      =     #Prozessdatenkanal_out.PO1_Steuerwort.reserve_15;
NETWORK
TITLE = Solldrehzahl
//Solldrehzahl (in 0,2 HZ) 
//== Sollfrequenz (in Hz) * 5 * Nenndrehzahl / Nennfrequenz
//
      L     #in_Sollfrequenz;
      L     #in_Motornenndrehzahl;
      *R;
      L     5.000000e+00;
      *R;
      L     #in_Motornennfrequenz;
      /R;
      T     #Solldrehzahl_tmp;	// (003)
      L     3.276700e+04;	// (003)
      >R;	// (003)
      JCN   SD_1;	// (003)
// maximale Drehzahl ausgeben wenn angeforderte größer als Maximalwert ist
      L     3.276700e+04;	// (003)
      RND;	// (003)
      T     #Prozessdatenkanal_out.PO2_Solldrehzahl;	// (003)
      JU    SD_L;	// (003)
// Drehzahl ausgeben wenn angeforderte kleiner als Maximalwert ist
SD_1: L     #Solldrehzahl_tmp;	// (003)
      RND;
      T     #Prozessdatenkanal_out.PO2_Solldrehzahl;
SD_L: AN    #in_Linkslauf;
      JC    E_SD;
      L     #Prozessdatenkanal_out.PO2_Solldrehzahl;
      L     -1;
      *I;
      T     #Prozessdatenkanal_out.PO2_Solldrehzahl;
E_SD: NOP   0;
NETWORK
TITLE = Warnungsbit
//(006) Netzwerk verschoben
//      U     #Prozessdatenkanal_in.PI1_Statuswort.Umrichter_betriebsbereit    // (004)
//      U     #Prozessdatenkanal_in.PI1_Statuswort.Stoerung_Warnung            // (004)
//      O                                        // (004)
      O(;	// (007)
      L     #Solldrehzahl_tmp;	// (006) #Prozessdatenkanal_out.PO2_Solldrehzahl    // (003)
      L     3.276700e+04;	// (003)
      >=R;	// (007)
      );	// (007)
      O(;	// (007)
      L     #Solldrehzahl_tmp;	// (006) #Prozessdatenkanal_out.PO2_Solldrehzahl    // (003)
      L     -3.276700e+04;	// (003)
      <=R;	// (007)
      );	// (007)
      =     #out_Warnung;
NETWORK
TITLE = Netzwerk für nicht unterstützte Funktionen
//Zur Standardisierung der E/A-Parameter aller FUs
      L     0.000000e+00;
      T     #out_Leistung;
      T     #out_Drehmoment;
      T     #out_Motorspannung;
NETWORK
TITLE = Daten an FU senden
// 8-Byte Parameterkanal
      CALL  "DPWR_DAT" (
           LADDR                    := #IO_Adr_Parameterkanal,
           RECORD                   := #Parameterkanal_out,
           RET_VAL                  := #Ret_Val_SFC15_1);
// 6-Byte Prozessdatenkanal
      CALL  "DPWR_DAT" (
           LADDR                    := #IO_Adr_Prozessdatenkanal,
           RECORD                   := #Prozessdatenkanal_out,
           RET_VAL                  := #Ret_Val_SFC15_2);
NETWORK
TITLE = Fehlercode L2Dp in FB_Fehlermeldung
      L     0;
      L     #Ret_Val_SFC14_1;
      <>I;
      JC    Fehl;
      L     0;
      L     #Ret_Val_SFC14_2;
      <>I;
      JC    Fehl;
      L     0;
      L     #Ret_Val_SFC15_1;
      <>I;
      JC    Fehl;
      L     0;
      L     #Ret_Val_SFC15_2;
      <>I;
      JC    Fehl;
      L     0;
Fehl: T     #out_FB_Fehlermeldung;
END_FUNCTION_BLOCK

FUNCTION_BLOCK "FB30 Daten von/an  FG"	// FB 30
TITLE = Ständiger Datenaustausch Visualisierung
//Erstellung:
//Datum        Bearbeiter                                                 Version
//--------------------------------------------------------------------------------
//00.00.00     Name (Kurzzeichen)                                         01.00.00
//
//Änderungen:
//Nr. Datum    Bearb Beschreibung                                   Marke Version
//--------------------------------------------------------------------------------
//01  25.01.17 gea   Automode = True; Manualmode = False            (001) 01.00.01
//
//03  15.01.2018 gea  expert service mode                           (003) 01.00.03
//
AUTHOR : sra
FAMILY : hsh
VERSION : 0.0
VAR
  reserve_IO : ARRAY  [0 .. 19 ] OF BYTE ;
  Datum_Uhrzeit_CPU : STRUCT
   von_Visualisierung : STRUCT
    set_actaul_date_time : BOOL ;
    set_date_and_time : STRUCT
     Jahr : BYTE ;
     Monat : BYTE ;
     Tag : BYTE ;
     Stunde : BYTE ;
     Minute : BYTE ;
     Sekunde : BYTE ;
     Millisekunde_H_Z : BYTE ;	//Millisekunden Hunderter und Zehnerstelle
     Millisekunde_E_Tag : BYTE ;	//Millisekunden Einerstelle und Wochentag (1=Sonntag)
    END_STRUCT ;
   END_STRUCT ;
   an_Visualisierung : STRUCT
    act_date_and_time : STRUCT
     Jahr : BYTE ;
     Monat : BYTE ;
     Tag : BYTE ;
     Stunde : BYTE ;
     Minute : BYTE ;
     Sekunde : BYTE ;
     Millisekunde_H_Z : BYTE ;	//Millisekunden Hunderter und Zehnerstelle
     Millisekunde_E_Tag : BYTE ;	//Millisekunden Einerstelle und Wochentag (1=Sonntag)
    END_STRUCT ;
   END_STRUCT ;
   reserve : ARRAY  [18 .. 19 ] OF BYTE ;
  END_STRUCT ;
  Watchdog : STRUCT
   Visualisierung : ARRAY  [1 .. 10 ] OF STRUCT
    von : INT ;
    an : INT ;
   END_STRUCT ;
   reserve_Watchdog : ARRAY  [40 .. 49 ] OF BYTE ;
  END_STRUCT ;
  Stoermeldung : STRUCT
   Steuerbits : STRUCT
    Quit_Sammelstoerung : BOOL ;
    reserve_0_1 : BOOL ;
    reserve_0_2 : BOOL ;
    reserve_0_3 : BOOL ;
    reserve_0_4 : BOOL ;
    reserve_0_5 : BOOL ;
    reserve_0_6 : BOOL ;
    reserve_0_7 : BOOL ;
   END_STRUCT ;
   Statusbits : STRUCT
    Sammelstoerung : BOOL ;
    reserve_0_1 : BOOL ;
    reserve_0_2 : BOOL ;
    reserve_0_3 : BOOL ;
    reserve_0_4 : BOOL ;
    reserve_0_5 : BOOL ;
    reserve_0_6 : BOOL ;
    reserve_0_7 : BOOL ;
   END_STRUCT ;
   reserve : ARRAY  [4 .. 9 ] OF BYTE ;
  END_STRUCT ;
  Anlage_ein_aus : STRUCT
   Anlagenbereich : ARRAY  [1 .. 10 ] OF STRUCT
    Steuerbits : STRUCT
     Anlage_ein : BOOL ;
     Anlage_aus : BOOL ;
     LampenTest : BOOL ;
     reserve_0_3 : BOOL ;
     reserve_0_4 : BOOL ;
     reserve_0_5 : BOOL ;
     reserve_0_6 : BOOL ;
     reserve_0_7 : BOOL ;
    END_STRUCT ;
    Statusbits : STRUCT
     Anlage_ein : BOOL ;	//1= Anlage ein
     Nothalt_OK : BOOL ;	//1= Nothalt OK (0= Anzeige blau)
     reserve_0_2 : BOOL ;
     simulationactive : BOOL ;
     reserve_0_4 : BOOL ;
     reserve_0_5 : BOOL ;
     reserve_0_6 : BOOL ;
     reserve_0_7 : BOOL ;
    END_STRUCT ;
   END_STRUCT ;
   reserve : ARRAY  [40 .. 99 ] OF BYTE ;
  END_STRUCT ;
  Modeschalter : STRUCT
   von_Visualisierung : STRUCT
    Servicemode_freigegeben : BOOL ;	//TRUE = Service Mode freigegeben
    ExpServicemode_freigegeb : BOOL ;	//TRUE = Service Mode freigegeben
    Automatikmode_Linie_Ber : ARRAY  [1 .. 64 ] OF //TRUE = Automode aktiv; FALSE= Manmode aktiv
    BOOL ;
    reserve : ARRAY  [10 .. 19 ] OF BYTE ;
   END_STRUCT ;
   an_Visualisierung : STRUCT
    Frg_Servicemode_ein : BOOL ;	//TRUE = Freigabe für Servicemodeumschaltung der Motor- und Ventilobjekte
    Frg_ExpService_mode_ein : BOOL ;	//TRUE = release service mode switch for motor and valve objects
    Anz_ExpService_mode_ein : BOOL ;	//TRUE = release service mode switch for motor and valve objects
    Frg_Hand_Auto_Linie_Ber : ARRAY  [1 .. 64 ] OF //TRUE=Frg für Umschaltung der Linie, Bereich, Mischer usw. von Hand auf Automode
    BOOL ;
    Frg_Auto_Hand_Linie_Ber : ARRAY  [1 .. 64 ] OF //TRUE=Frg für Umschaltung der Linie, Bereich, Mischer usw. von Auto auf Handmode
    BOOL ;
    Ursache_gesperrt : STRUCT 	//Ursache für das Sperren des Modeschalters (optional)
     Servicemode : INT ;
     Hand_Auto : ARRAY  [1 .. 64 ] OF INT ;
    END_STRUCT ;
   END_STRUCT ;
   reserve : ARRAY  [168 .. 199 ] OF BYTE ;
  END_STRUCT ;
  allgemeine_Signale : STRUCT
   Lampentest : BOOL ;
   reserve : ARRAY  [2 .. 99 ] OF BYTE ;
  END_STRUCT ;
END_VAR
VAR_TEMP
  set_date_and_time : DATE_AND_TIME ;
  act_date_and_time : DATE_AND_TIME ;
  Ret_Val_SFC0_SFC1 : INT ;
END_VAR
BEGIN
NETWORK
TITLE = Datum und Uhrzeit schreiben
//Wandlung von Integer in BCD-Format 
      AN    #Datum_Uhrzeit_CPU.von_Visualisierung.set_actaul_date_time;
      JC    E_DT;
      LAR1  P##set_date_and_time;
      L     #Datum_Uhrzeit_CPU.von_Visualisierung.set_date_and_time.Jahr;
//      ITB                               // wird bei Projekten im TIA-Portal nicht benötigt
      T     LB [AR1,P#0.0];
      L     #Datum_Uhrzeit_CPU.von_Visualisierung.set_date_and_time.Monat;
//      ITB                               // wird bei Projekten im TIA-Portal nicht benötigt
      T     LB [AR1,P#1.0];
      L     #Datum_Uhrzeit_CPU.von_Visualisierung.set_date_and_time.Tag;
//      ITB                               // wird bei Projekten im TIA-Portal nicht benötigt
      T     LB [AR1,P#2.0];
      L     #Datum_Uhrzeit_CPU.von_Visualisierung.set_date_and_time.Stunde;
//      ITB                               // wird bei Projekten im TIA-Portal nicht benötigt
      T     LB [AR1,P#3.0];
      L     #Datum_Uhrzeit_CPU.von_Visualisierung.set_date_and_time.Minute;
//      ITB                               // wird bei Projekten im TIA-Portal nicht benötigt
      T     LB [AR1,P#4.0];
      L     #Datum_Uhrzeit_CPU.von_Visualisierung.set_date_and_time.Sekunde;
//      ITB                               // wird bei Projekten im TIA-Portal nicht benötigt
      T     LB [AR1,P#5.0];
      L     #Datum_Uhrzeit_CPU.von_Visualisierung.set_date_and_time.Millisekunde_H_Z;
//      ITB                               // wird bei Projekten im TIA-Portal nicht benötigt
      T     LB [AR1,P#6.0];
      L     #Datum_Uhrzeit_CPU.von_Visualisierung.set_date_and_time.Millisekunde_E_Tag;
//      ITB                               // wird bei Projekten im TIA-Portal nicht benötigt
      T     LB [AR1,P#7.0];
      CALL  "SET_CLK" (
           PDT                      := #set_date_and_time,
           RET_VAL                  := #Ret_Val_SFC0_SFC1);
      SET;
      R     #Datum_Uhrzeit_CPU.von_Visualisierung.set_actaul_date_time;
E_DT: NOP   0;
NETWORK
TITLE = Datum und Uhrzeit lesen
//read date and time 
      CALL  "READ_CLK" (
           RET_VAL                  := #Ret_Val_SFC0_SFC1,
           CDT                      := #act_date_and_time);
NETWORK
TITLE = aktuelles Datum und Uhrzeit wandeln 
//Wandlung von BCD_Format in Integer
      LAR1  P##act_date_and_time;
      L     LB [AR1,P#0.0];
//      BTI                               // wird bei Projekten im TIA-Portal nicht benötigt
      T     #Datum_Uhrzeit_CPU.an_Visualisierung.act_date_and_time.Jahr;
      L     LB [AR1,P#1.0];
//      BTI                               // wird bei Projekten im TIA-Portal nicht benötigt
      T     #Datum_Uhrzeit_CPU.an_Visualisierung.act_date_and_time.Monat;
      L     LB [AR1,P#2.0];
//      BTI                               // wird bei Projekten im TIA-Portal nicht benötigt
      T     #Datum_Uhrzeit_CPU.an_Visualisierung.act_date_and_time.Tag;
      L     LB [AR1,P#3.0];
//      BTI                               // wird bei Projekten im TIA-Portal nicht benötigt
      T     #Datum_Uhrzeit_CPU.an_Visualisierung.act_date_and_time.Stunde;
      L     LB [AR1,P#4.0];
//      BTI                               // wird bei Projekten im TIA-Portal nicht benötigt
      T     #Datum_Uhrzeit_CPU.an_Visualisierung.act_date_and_time.Minute;
      L     LB [AR1,P#5.0];
//      BTI                               // wird bei Projekten im TIA-Portal nicht benötigt
      T     #Datum_Uhrzeit_CPU.an_Visualisierung.act_date_and_time.Sekunde;
      L     LB [AR1,P#6.0];
//      BTI                               // wird bei Projekten im TIA-Portal nicht benötigt
      T     #Datum_Uhrzeit_CPU.an_Visualisierung.act_date_and_time.Millisekunde_H_Z;
      L     LB [AR1,P#7.0];
//      BTI                               // wird bei Projekten im TIA-Portal nicht benötigt
      T     #Datum_Uhrzeit_CPU.an_Visualisierung.act_date_and_time.Millisekunde_E_Tag;
NETWORK
TITLE = ------------  Watchdog ----------------------
NETWORK
TITLE = Watchdog Visualisierung
//je ein Watchdog pro PC
      L     #Watchdog.Visualisierung[1].von;
      T     #Watchdog.Visualisierung[1].an;
NETWORK
TITLE = ------------  Sammelstörung ----------------------
NETWORK
TITLE = Sammelstörung und Quittierung
      A     #Stoermeldung.Steuerbits.Quit_Sammelstoerung;
      =     "M1.0 AcknowledgeFault";
      A     "M1.1 Fault(General)";
      =     #Stoermeldung.Statusbits.Sammelstoerung;
      =     "Q 5.1";
NETWORK
TITLE = ------------  Lampentest ----------------------
NETWORK
TITLE = global lamp testing
      A     #Anlage_ein_aus.Anlagenbereich[1].Steuerbits.LampenTest;
      =     "GlobalLampTesting";
NETWORK
TITLE = ------------  Motor/Ventil Handling  ----------------------
NETWORK
TITLE = Simulation active
      A     "M0.5 SimulationInternal";
      =     #Anlage_ein_aus.Anlagenbereich[1].Statusbits.simulationactive;
NETWORK
TITLE = Freigabesignale für Kontrollmodule
      A     #Modeschalter.von_Visualisierung.Servicemode_freigegeben;
      =     "Release Man Mode Motors";
      =     "Release Man Mode Valves";
// define if fault messages of motors has to be acknowledged
      SET;
      =     "AckObligatoryMotors";
// define if fault messages of flaps has to be acknowledged
      CLR;
      =     "AckObligatoryValves";
NETWORK
TITLE = Service Mode (Motor + Ventile)
//Service Mode zentral sperren
      AN    #Modeschalter.von_Visualisierung.Servicemode_freigegeben;
      =     "M0.0 LockManualMode";
//Freigabe für Service Mode Schalter aus SPS
      SET;
      =     #Modeschalter.an_Visualisierung.Frg_Servicemode_ein;
NETWORK
TITLE = Expert Service mode
//(003)
      A     #Modeschalter.von_Visualisierung.Servicemode_freigegeben;
      =     "Service Mode ExpertMode";
      SET;
      =     #Modeschalter.an_Visualisierung.Frg_ExpService_mode_ein;
      SET;
      =     #Modeschalter.an_Visualisierung.Anz_ExpService_mode_ein;
NETWORK
TITLE = ------------- System on/off --------------
NETWORK
TITLE = Nothalt (Anlagenbereich 1)
      A     "I 5.2";	// Eingang "Nothalt OK" Anlagenbereich 1
      SET;	// no NH
      =     #Anlage_ein_aus.Anlagenbereich[1].Statusbits.Nothalt_OK;
NETWORK
TITLE = Anlage ein (Anlagenbereich 1)
//Jeder Anlagenbereich ist separat ein- und ausschaltbar. 
//Beim Betätigen des Not-Halt Schalters 
      A     #Anlage_ein_aus.Anlagenbereich[1].Steuerbits.Anlage_ein;
//     O     "I 5.0"                     // taste ON
//    A     #Anlage_ein_aus.Anlagenbereich[1].Statusbits.Nothalt_OK    // Eingang "Nothalt OK" Anlagenbereich 1
      S     #Anlage_ein_aus.Anlagenbereich[1].Statusbits.Anlage_ein;
      O     #Anlage_ein_aus.Anlagenbereich[1].Steuerbits.Anlage_aus;
//    O     "02_01_101_Gp"              //tatse off
//      ON    #Anlage_ein_aus.Anlagenbereich[1].Statusbits.Nothalt_OK    // Eingang "Nothalt OK" Anlagenbereich 1
      R     #Anlage_ein_aus.Anlagenbereich[1].Statusbits.Anlage_ein;
      AN    #Anlage_ein_aus.Anlagenbereich[1].Statusbits.Anlage_ein;
      =     DB34.DBX 205.0;
NETWORK
TITLE = Lampe Anlage ein (Anlagenbereich 1)
//  A     #Anlage_ein_aus.Anlagenbereich[1].Statusbits.Anlage_ein
//      =     "Q 5.0"                     // Ausgang "Anlage ein" Anlagenbereich 1
NETWORK
TITLE = Nothalt (Anlagenbereich 2)
//// No 2 nd Area
//    A     I      0.1                  // Eingang "Nothalt OK" Anlagenbereich 2
//      =     #Anlage_ein_aus.Anlagenbereich[2].Statusbits.Nothalt_OK
NETWORK
TITLE = Anlage ein (Anlagenbereich 2)
// // No 2 nd Area
//      A     #Anlage_ein_aus.Anlagenbereich[2].Steuerbits.Anlage_ein
//      A     #Anlage_ein_aus.Anlagenbereich[2].Statusbits.Nothalt_OK    // Eingang "Nothalt OK" Anlagenbereich 2
//      S     #Anlage_ein_aus.Anlagenbereich[2].Statusbits.Anlage_ein
//      O     #Anlage_ein_aus.Anlagenbereich[2].Steuerbits.Anlage_aus
//      ON    #Anlage_ein_aus.Anlagenbereich[2].Statusbits.Nothalt_OK    // Eingang "Nothalt OK" Anlagenbereich 2
//      R     #Anlage_ein_aus.Anlagenbereich[2].Statusbits.Anlage_ein
NETWORK
TITLE = Lampe Anlage ein (Anlagenbereich 2)
//      A     #Anlage_ein_aus.Anlagenbereich[2].Statusbits.Anlage_ein
//      =     Q      0.1                  // Ausgang "Anlage ein" Anlagenbereich 2
NETWORK
TITLE = Freigabe Modeschalter
// No scales. no mixers
// Umschaltung von Automatikmode auf Handmode ist immer freigegeben
//      A     #Modeschalter.von_Visualisierung.Automatikmode_Linie_Ber[1]    //(001)
//      =     #Modeschalter.an_Visualisierung.Frg_Auto_Hand_Linie_Ber[1]
// Umschaltung von Handmode auf Automatikmode ist freigegeben freigegeben wenn alle Anlagenteile im Grundzustand und leer sind
//      AN    #Modeschalter.von_Visualisierung.Automatikmode_Linie_Ber[1]    //(001)
//    U     alle Waagen im Grundzustand
//    U     alle Waagen leer
//    U     Mischer im Automatikmode
//      =     #Modeschalter.an_Visualisierung.Frg_Hand_Auto_Linie_Ber[1]
NETWORK
TITLE = Ursache für Modeschalter 1 gesperrt
//0:         Leerer Text, nicht definiert
//1..100:    Waage nicht und leer
//            1 = Waage 1, 2 = Waage 2 usw.
//101..200:  Waage nicht befüllt (Negativwaage)
//            101 = Waage 1, 102 = Waage 2 usw.
//201..300:  Mischer (Heizmischer) nicht leer
//            201 = Mischer 1, 202 = Mischer 2
//301..400:  Mischer (Kühlmischer) nicht leer
//            301 = Mischer 1, 302 = Mischer 2
//401..500:  Waage nicht in Grundzustand
//            401 = Waage 1, 402 = Waage 2 usw.
//501..600:  Waage meldet Fehler
//            501 = Waage 1, 502 = Waage 2 usw.
//
//
//
////  No mix/scales - >> commented
//
// Beispiel für Modeschalter 1
//      AN    #Modeschalter.von_Visualisierung.Automatikmode_Linie_Ber[1]    //(001)
//      JC    L1OK
//    ON   Waage_1_leer
//      L     1
//      JC    SL_1
//    ON   Waage_2_leer
//      L     2
//      JC    SL_1
//    :
//    O    Waage_5_nicht_befuellt
//      L     105
//      JC    SL_1
//    :
//    ON   Mischer_1_leer
//      L     201
//      JC    SL_1
//    ON  Waage_1_im_Grundzustand
//      L     401
//      JC    SL_1
//L1OK: L     0
//SL_1: T     #Modeschalter.an_Visualisierung.Ursache_gesperrt.Hand_Auto[1]
END_FUNCTION_BLOCK

FUNCTION_BLOCK "FB31 Mode Objekte an FG"	// FB 31
TITLE = Handbetrieb an Farbgrafik
//Erstellung:
//Datum        Bearbeiter                                                 Version
//--------------------------------------------------------------------------------
//00.00.00     xxx                                                        01.00.00
//
//Änderungen:
//Nr. Datum    Bearb Beschreibung                                   Marke Version
//--------------------------------------------------------------------------------
//01  00.00.00                                                      (xxx) xx.xx.xx
//
//--------------------------------------------------------------------------------
//
//
AUTHOR : sra
FAMILY : SCADA
NAME : mode
VERSION : 0.0
VAR
  Auto_Handmode_A : ARRAY  [0 .. 128, 0 .. 7 ] OF BOOL ;
END_VAR
BEGIN
NETWORK
TITLE = Handbetrieb Objekt 1
//      U     DBxyz.DBX  x.y
//      =     #Auto_Handmode_A[x, y]
NETWORK
TITLE =
END_FUNCTION_BLOCK

FUNCTION_BLOCK "FB32 Eingaege an FG"	// FB 32
TITLE = Eingänge für Farbgrafik in Datenworte des DB32 speichern
//Erstellung:
//Datum        Bearbeiter                                                 Version
//--------------------------------------------------------------------------------
//00.00.00     xxx                                                        01.00.00
//
//Änderungen:
//Nr. Datum    Bearb Beschreibung                                   Marke Version
//--------------------------------------------------------------------------------
//01  00.00.00                                                      (xxx) xx.xx.xx
//
//--------------------------------------------------------------------------------
//
//
AUTHOR : sra
FAMILY : SCADA
NAME : inputs
VERSION : 0.0
VAR
  input_0_0 : BOOL ;
  input_0_1 : BOOL ;
  input_0_2 : BOOL ;
  input_0_3 : BOOL ;
  input_0_4 : BOOL ;
  input_0_5 : BOOL ;
  input_0_6 : BOOL ;
  input_0_7 : BOOL ;
  input_1_0 : BOOL ;
  input_1_1 : BOOL ;
  input_1_2 : BOOL ;
  input_1_3 : BOOL ;
  input_1_4 : BOOL ;
  input_1_5 : BOOL ;
  input_1_6 : BOOL ;
  input_1_7 : BOOL ;
  input_2_0 : BOOL ;
  input_2_1 : BOOL ;
  input_2_2 : BOOL ;
  input_2_3 : BOOL ;
  input_2_4 : BOOL ;
  input_2_5 : BOOL ;
  input_2_6 : BOOL ;
  input_2_7 : BOOL ;
  input_3_0 : BOOL ;
  input_3_1 : BOOL ;
  input_3_2 : BOOL ;
  input_3_3 : BOOL ;
  input_3_4 : BOOL ;
  input_3_5 : BOOL ;
  input_3_6 : BOOL ;
  input_3_7 : BOOL ;
  input_4_0 : BOOL ;
  input_4_1 : BOOL ;
  input_4_2 : BOOL ;
  input_4_3 : BOOL ;
  input_4_4 : BOOL ;
  input_4_5 : BOOL ;
  input_4_6 : BOOL ;
  input_4_7 : BOOL ;
  input_5_0 : BOOL ;
  input_5_1 : BOOL ;
  input_5_2 : BOOL ;
  input_5_3 : BOOL ;
  input_5_4 : BOOL ;
  input_5_5 : BOOL ;
  input_5_6 : BOOL ;
  input_5_7 : BOOL ;
  input_6_0 : BOOL ;
  input_6_1 : BOOL ;
  input_6_2 : BOOL ;
  input_6_3 : BOOL ;
  input_6_4 : BOOL ;
  input_6_5 : BOOL ;
  input_6_6 : BOOL ;
  input_6_7 : BOOL ;
  input_7_0 : BOOL ;
  input_7_1 : BOOL ;
  input_7_2 : BOOL ;
  input_7_3 : BOOL ;
  input_7_4 : BOOL ;
  input_7_5 : BOOL ;
  input_7_6 : BOOL ;
  input_7_7 : BOOL ;
  input_8_0 : BOOL ;
  input_8_1 : BOOL ;
  input_8_2 : BOOL ;
  input_8_3 : BOOL ;
  input_8_4 : BOOL ;
  input_8_5 : BOOL ;
  input_8_6 : BOOL ;
  input_8_7 : BOOL ;
  input_9_0 : BOOL ;
  input_9_1 : BOOL ;
  input_9_2 : BOOL ;
  input_9_3 : BOOL ;
  input_9_4 : BOOL ;
  input_9_5 : BOOL ;
  input_9_6 : BOOL ;
  input_9_7 : BOOL ;
  input_10_0 : BOOL ;
  input_10_1 : BOOL ;
  input_10_2 : BOOL ;
  input_10_3 : BOOL ;
  input_10_4 : BOOL ;
  input_10_5 : BOOL ;
  input_10_6 : BOOL ;
  input_10_7 : BOOL ;
  input_11_0 : BOOL ;
  input_11_1 : BOOL ;
  input_11_2 : BOOL ;
  input_11_3 : BOOL ;
  input_11_4 : BOOL ;
  input_11_5 : BOOL ;
  input_11_6 : BOOL ;
  input_11_7 : BOOL ;
  input_12_0 : BOOL ;
  input_12_1 : BOOL ;
  input_12_2 : BOOL ;
  input_12_3 : BOOL ;
  input_12_4 : BOOL ;
  input_12_5 : BOOL ;
  input_12_6 : BOOL ;
  input_12_7 : BOOL ;
  input_13_0 : BOOL ;
  input_13_1 : BOOL ;
  input_13_2 : BOOL ;
  input_13_3 : BOOL ;
  input_13_4 : BOOL ;
  input_13_5 : BOOL ;
  input_13_6 : BOOL ;
  input_13_7 : BOOL ;
  input_14_0 : BOOL ;
  input_14_1 : BOOL ;
  input_14_2 : BOOL ;
  input_14_3 : BOOL ;
  input_14_4 : BOOL ;
  input_14_5 : BOOL ;
  input_14_6 : BOOL ;
  input_14_7 : BOOL ;
  input_15_0 : BOOL ;
  input_15_1 : BOOL ;
  input_15_2 : BOOL ;
  input_15_3 : BOOL ;
  input_15_4 : BOOL ;
  input_15_5 : BOOL ;
  input_15_6 : BOOL ;
  input_15_7 : BOOL ;
  input_16_0 : BOOL ;
  input_16_1 : BOOL ;
  input_16_2 : BOOL ;
  input_16_3 : BOOL ;
  input_16_4 : BOOL ;
  input_16_5 : BOOL ;
  input_16_6 : BOOL ;
  input_16_7 : BOOL ;
  input_17_0 : BOOL ;
  input_17_1 : BOOL ;
  input_17_2 : BOOL ;
  input_17_3 : BOOL ;
  input_17_4 : BOOL ;
  input_17_5 : BOOL ;
  input_17_6 : BOOL ;
  input_17_7 : BOOL ;
  input_18_0 : BOOL ;
  input_18_1 : BOOL ;
  input_18_2 : BOOL ;
  input_18_3 : BOOL ;
  input_18_4 : BOOL ;
  input_18_5 : BOOL ;
  input_18_6 : BOOL ;
  input_18_7 : BOOL ;
  input_19_0 : BOOL ;
  input_19_1 : BOOL ;
  input_19_2 : BOOL ;
  input_19_3 : BOOL ;
  input_19_4 : BOOL ;
  input_19_5 : BOOL ;
  input_19_6 : BOOL ;
  input_19_7 : BOOL ;
  input_20_0 : BOOL ;
  input_20_1 : BOOL ;
  input_20_2 : BOOL ;
  input_20_3 : BOOL ;
  input_20_4 : BOOL ;
  input_20_5 : BOOL ;
  input_20_6 : BOOL ;
  input_20_7 : BOOL ;
  input_21_0 : BOOL ;
  input_21_1 : BOOL ;
  input_21_2 : BOOL ;
  input_21_3 : BOOL ;
  input_21_4 : BOOL ;
  input_21_5 : BOOL ;
  input_21_6 : BOOL ;
  input_21_7 : BOOL ;
  input_22_0 : BOOL ;
  input_22_1 : BOOL ;
  input_22_2 : BOOL ;
  input_22_3 : BOOL ;
  input_22_4 : BOOL ;
  input_22_5 : BOOL ;
  input_22_6 : BOOL ;
  input_22_7 : BOOL ;
  input_23_0 : BOOL ;
  input_23_1 : BOOL ;
  input_23_2 : BOOL ;
  input_23_3 : BOOL ;
  input_23_4 : BOOL ;
  input_23_5 : BOOL ;
  input_23_6 : BOOL ;
  input_23_7 : BOOL ;
  input_24_0 : BOOL ;
  input_24_1 : BOOL ;
  input_24_2 : BOOL ;
  input_24_3 : BOOL ;
  input_24_4 : BOOL ;
  input_24_5 : BOOL ;
  input_24_6 : BOOL ;
  input_24_7 : BOOL ;
  input_25_0 : BOOL ;
  input_25_1 : BOOL ;
  input_25_2 : BOOL ;
  input_25_3 : BOOL ;
  input_25_4 : BOOL ;
  input_25_5 : BOOL ;
  input_25_6 : BOOL ;
  input_25_7 : BOOL ;
  input_26_0 : BOOL ;
  input_26_1 : BOOL ;
  input_26_2 : BOOL ;
  input_26_3 : BOOL ;
  input_26_4 : BOOL ;
  input_26_5 : BOOL ;
  input_26_6 : BOOL ;
  input_26_7 : BOOL ;
  input_27_0 : BOOL ;
  input_27_1 : BOOL ;
  input_27_2 : BOOL ;
  input_27_3 : BOOL ;
  input_27_4 : BOOL ;
  input_27_5 : BOOL ;
  input_27_6 : BOOL ;
  input_27_7 : BOOL ;
  input_28_0 : BOOL ;
  input_28_1 : BOOL ;
  input_28_2 : BOOL ;
  input_28_3 : BOOL ;
  input_28_4 : BOOL ;
  input_28_5 : BOOL ;
  input_28_6 : BOOL ;
  input_28_7 : BOOL ;
  input_29_0 : BOOL ;
  input_29_1 : BOOL ;
  input_29_2 : BOOL ;
  input_29_3 : BOOL ;
  input_29_4 : BOOL ;
  input_29_5 : BOOL ;
  input_29_6 : BOOL ;
  input_29_7 : BOOL ;
  input_30_0 : BOOL ;
  input_30_1 : BOOL ;
  input_30_2 : BOOL ;
  input_30_3 : BOOL ;
  input_30_4 : BOOL ;
  input_30_5 : BOOL ;
  input_30_6 : BOOL ;
  input_30_7 : BOOL ;
  input_31_0 : BOOL ;
  input_31_1 : BOOL ;
  input_31_2 : BOOL ;
  input_31_3 : BOOL ;
  input_31_4 : BOOL ;
  input_31_5 : BOOL ;
  input_31_6 : BOOL ;
  input_31_7 : BOOL ;
  input_32_0 : BOOL ;
  input_32_1 : BOOL ;
  input_32_2 : BOOL ;
  input_32_3 : BOOL ;
  input_32_4 : BOOL ;
  input_32_5 : BOOL ;
  input_32_6 : BOOL ;
  input_32_7 : BOOL ;
  input_33_0 : BOOL ;
  input_33_1 : BOOL ;
  input_33_2 : BOOL ;
  input_33_3 : BOOL ;
  input_33_4 : BOOL ;
  input_33_5 : BOOL ;
  input_33_6 : BOOL ;
  input_33_7 : BOOL ;
  input_34_0 : BOOL ;
  input_34_1 : BOOL ;
  input_34_2 : BOOL ;
  input_34_3 : BOOL ;
  input_34_4 : BOOL ;
  input_34_5 : BOOL ;
  input_34_6 : BOOL ;
  input_34_7 : BOOL ;
  input_35_0 : BOOL ;
  input_35_1 : BOOL ;
  input_35_2 : BOOL ;
  input_35_3 : BOOL ;
  input_35_4 : BOOL ;
  input_35_5 : BOOL ;
  input_35_6 : BOOL ;
  input_35_7 : BOOL ;
  input_36_0 : BOOL ;
  input_36_1 : BOOL ;
  input_36_2 : BOOL ;
  input_36_3 : BOOL ;
  input_36_4 : BOOL ;
  input_36_5 : BOOL ;
  input_36_6 : BOOL ;
  input_36_7 : BOOL ;
  input_37_0 : BOOL ;
  input_37_1 : BOOL ;
  input_37_2 : BOOL ;
  input_37_3 : BOOL ;
  input_37_4 : BOOL ;
  input_37_5 : BOOL ;
  input_37_6 : BOOL ;
  input_37_7 : BOOL ;
  input_38_0 : BOOL ;
  input_38_1 : BOOL ;
  input_38_2 : BOOL ;
  input_38_3 : BOOL ;
  input_38_4 : BOOL ;
  input_38_5 : BOOL ;
  input_38_6 : BOOL ;
  input_38_7 : BOOL ;
  input_39_0 : BOOL ;
  input_39_1 : BOOL ;
  input_39_2 : BOOL ;
  input_39_3 : BOOL ;
  input_39_4 : BOOL ;
  input_39_5 : BOOL ;
  input_39_6 : BOOL ;
  input_39_7 : BOOL ;
  input_40_0 : BOOL ;
  input_40_1 : BOOL ;
  input_40_2 : BOOL ;
  input_40_3 : BOOL ;
  input_40_4 : BOOL ;
  input_40_5 : BOOL ;
  input_40_6 : BOOL ;
  input_40_7 : BOOL ;
  input_41_0 : BOOL ;
  input_41_1 : BOOL ;
  input_41_2 : BOOL ;
  input_41_3 : BOOL ;
  input_41_4 : BOOL ;
  input_41_5 : BOOL ;
  input_41_6 : BOOL ;
  input_41_7 : BOOL ;
  input_42_0 : BOOL ;
  input_42_1 : BOOL ;
  input_42_2 : BOOL ;
  input_42_3 : BOOL ;
  input_42_4 : BOOL ;
  input_42_5 : BOOL ;
  input_42_6 : BOOL ;
  input_42_7 : BOOL ;
  input_43_0 : BOOL ;
  input_43_1 : BOOL ;
  input_43_2 : BOOL ;
  input_43_3 : BOOL ;
  input_43_4 : BOOL ;
  input_43_5 : BOOL ;
  input_43_6 : BOOL ;
  input_43_7 : BOOL ;
  input_44_0 : BOOL ;
  input_44_1 : BOOL ;
  input_44_2 : BOOL ;
  input_44_3 : BOOL ;
  input_44_4 : BOOL ;
  input_44_5 : BOOL ;
  input_44_6 : BOOL ;
  input_44_7 : BOOL ;
  input_45_0 : BOOL ;
  input_45_1 : BOOL ;
  input_45_2 : BOOL ;
  input_45_3 : BOOL ;
  input_45_4 : BOOL ;
  input_45_5 : BOOL ;
  input_45_6 : BOOL ;
  input_45_7 : BOOL ;
  input_46_0 : BOOL ;
  input_46_1 : BOOL ;
  input_46_2 : BOOL ;
  input_46_3 : BOOL ;
  input_46_4 : BOOL ;
  input_46_5 : BOOL ;
  input_46_6 : BOOL ;
  input_46_7 : BOOL ;
  input_47_0 : BOOL ;
  input_47_1 : BOOL ;
  input_47_2 : BOOL ;
  input_47_3 : BOOL ;
  input_47_4 : BOOL ;
  input_47_5 : BOOL ;
  input_47_6 : BOOL ;
  input_47_7 : BOOL ;
  input_48_0 : BOOL ;
  input_48_1 : BOOL ;
  input_48_2 : BOOL ;
  input_48_3 : BOOL ;
  input_48_4 : BOOL ;
  input_48_5 : BOOL ;
  input_48_6 : BOOL ;
  input_48_7 : BOOL ;
  input_49_0 : BOOL ;
  input_49_1 : BOOL ;
  input_49_2 : BOOL ;
  input_49_3 : BOOL ;
  input_49_4 : BOOL ;
  input_49_5 : BOOL ;
  input_49_6 : BOOL ;
  input_49_7 : BOOL ;
  input_50_0 : BOOL ;
  input_50_1 : BOOL ;
  input_50_2 : BOOL ;
  input_50_3 : BOOL ;
  input_50_4 : BOOL ;
  input_50_5 : BOOL ;
  input_50_6 : BOOL ;
  input_50_7 : BOOL ;
  input_51_0 : BOOL ;
  input_51_1 : BOOL ;
  input_51_2 : BOOL ;
  input_51_3 : BOOL ;
  input_51_4 : BOOL ;
  input_51_5 : BOOL ;
  input_51_6 : BOOL ;
  input_51_7 : BOOL ;
  input_52_0 : BOOL ;
  input_52_1 : BOOL ;
  input_52_2 : BOOL ;
  input_52_3 : BOOL ;
  input_52_4 : BOOL ;
  input_52_5 : BOOL ;
  input_52_6 : BOOL ;
  input_52_7 : BOOL ;
  input_53_0 : BOOL ;
  input_53_1 : BOOL ;
  input_53_2 : BOOL ;
  input_53_3 : BOOL ;
  input_53_4 : BOOL ;
  input_53_5 : BOOL ;
  input_53_6 : BOOL ;
  input_53_7 : BOOL ;
  input_54_0 : BOOL ;
  input_54_1 : BOOL ;
  input_54_2 : BOOL ;
  input_54_3 : BOOL ;
  input_54_4 : BOOL ;
  input_54_5 : BOOL ;
  input_54_6 : BOOL ;
  input_54_7 : BOOL ;
  input_55_0 : BOOL ;
  input_55_1 : BOOL ;
  input_55_2 : BOOL ;
  input_55_3 : BOOL ;
  input_55_4 : BOOL ;
  input_55_5 : BOOL ;
  input_55_6 : BOOL ;
  input_55_7 : BOOL ;
  input_56_0 : BOOL ;
  input_56_1 : BOOL ;
  input_56_2 : BOOL ;
  input_56_3 : BOOL ;
  input_56_4 : BOOL ;
  input_56_5 : BOOL ;
  input_56_6 : BOOL ;
  input_56_7 : BOOL ;
  input_57_0 : BOOL ;
  input_57_1 : BOOL ;
  input_57_2 : BOOL ;
  input_57_3 : BOOL ;
  input_57_4 : BOOL ;
  input_57_5 : BOOL ;
  input_57_6 : BOOL ;
  input_57_7 : BOOL ;
  input_58_0 : BOOL ;
  input_58_1 : BOOL ;
  input_58_2 : BOOL ;
  input_58_3 : BOOL ;
  input_58_4 : BOOL ;
  input_58_5 : BOOL ;
  input_58_6 : BOOL ;
  input_58_7 : BOOL ;
  input_59_0 : BOOL ;
  input_59_1 : BOOL ;
  input_59_2 : BOOL ;
  input_59_3 : BOOL ;
  input_59_4 : BOOL ;
  input_59_5 : BOOL ;
  input_59_6 : BOOL ;
  input_59_7 : BOOL ;
  input_60_0 : BOOL ;
  input_60_1 : BOOL ;
  input_60_2 : BOOL ;
  input_60_3 : BOOL ;
  input_60_4 : BOOL ;
  input_60_5 : BOOL ;
  input_60_6 : BOOL ;
  input_60_7 : BOOL ;
  input_61_0 : BOOL ;
  input_61_1 : BOOL ;
  input_61_2 : BOOL ;
  input_61_3 : BOOL ;
  input_61_4 : BOOL ;
  input_61_5 : BOOL ;
  input_61_6 : BOOL ;
  input_61_7 : BOOL ;
  input_62_0 : BOOL ;
  input_62_1 : BOOL ;
  input_62_2 : BOOL ;
  input_62_3 : BOOL ;
  input_62_4 : BOOL ;
  input_62_5 : BOOL ;
  input_62_6 : BOOL ;
  input_62_7 : BOOL ;
  input_63_0 : BOOL ;
  input_63_1 : BOOL ;
  input_63_2 : BOOL ;
  input_63_3 : BOOL ;
  input_63_4 : BOOL ;
  input_63_5 : BOOL ;
  input_63_6 : BOOL ;
  input_63_7 : BOOL ;
  input_64_0 : BOOL ;
  input_64_1 : BOOL ;
  input_64_2 : BOOL ;
  input_64_3 : BOOL ;
  input_64_4 : BOOL ;
  input_64_5 : BOOL ;
  input_64_6 : BOOL ;
  input_64_7 : BOOL ;
  input_65_0 : BOOL ;
  input_65_1 : BOOL ;
  input_65_2 : BOOL ;
  input_65_3 : BOOL ;
  input_65_4 : BOOL ;
  input_65_5 : BOOL ;
  input_65_6 : BOOL ;
  input_65_7 : BOOL ;
  input_66_0 : BOOL ;
  input_66_1 : BOOL ;
  input_66_2 : BOOL ;
  input_66_3 : BOOL ;
  input_66_4 : BOOL ;
  input_66_5 : BOOL ;
  input_66_6 : BOOL ;
  input_66_7 : BOOL ;
  input_67_0 : BOOL ;
  input_67_1 : BOOL ;
  input_67_2 : BOOL ;
  input_67_3 : BOOL ;
  input_67_4 : BOOL ;
  input_67_5 : BOOL ;
  input_67_6 : BOOL ;
  input_67_7 : BOOL ;
  input_68_0 : BOOL ;
  input_68_1 : BOOL ;
  input_68_2 : BOOL ;
  input_68_3 : BOOL ;
  input_68_4 : BOOL ;
  input_68_5 : BOOL ;
  input_68_6 : BOOL ;
  input_68_7 : BOOL ;
  input_69_0 : BOOL ;
  input_69_1 : BOOL ;
  input_69_2 : BOOL ;
  input_69_3 : BOOL ;
  input_69_4 : BOOL ;
  input_69_5 : BOOL ;
  input_69_6 : BOOL ;
  input_69_7 : BOOL ;
  input_70_0 : BOOL ;
  input_70_1 : BOOL ;
  input_70_2 : BOOL ;
  input_70_3 : BOOL ;
  input_70_4 : BOOL ;
  input_70_5 : BOOL ;
  input_70_6 : BOOL ;
  input_70_7 : BOOL ;
  input_71_0 : BOOL ;
  input_71_1 : BOOL ;
  input_71_2 : BOOL ;
  input_71_3 : BOOL ;
  input_71_4 : BOOL ;
  input_71_5 : BOOL ;
  input_71_6 : BOOL ;
  input_71_7 : BOOL ;
  input_72_0 : BOOL ;
  input_72_1 : BOOL ;
  input_72_2 : BOOL ;
  input_72_3 : BOOL ;
  input_72_4 : BOOL ;
  input_72_5 : BOOL ;
  input_72_6 : BOOL ;
  input_72_7 : BOOL ;
  input_73_0 : BOOL ;
  input_73_1 : BOOL ;
  input_73_2 : BOOL ;
  input_73_3 : BOOL ;
  input_73_4 : BOOL ;
  input_73_5 : BOOL ;
  input_73_6 : BOOL ;
  input_73_7 : BOOL ;
  input_74_0 : BOOL ;
  input_74_1 : BOOL ;
  input_74_2 : BOOL ;
  input_74_3 : BOOL ;
  input_74_4 : BOOL ;
  input_74_5 : BOOL ;
  input_74_6 : BOOL ;
  input_74_7 : BOOL ;
  input_75_0 : BOOL ;
  input_75_1 : BOOL ;
  input_75_2 : BOOL ;
  input_75_3 : BOOL ;
  input_75_4 : BOOL ;
  input_75_5 : BOOL ;
  input_75_6 : BOOL ;
  input_75_7 : BOOL ;
  input_76_0 : BOOL ;
  input_76_1 : BOOL ;
  input_76_2 : BOOL ;
  input_76_3 : BOOL ;
  input_76_4 : BOOL ;
  input_76_5 : BOOL ;
  input_76_6 : BOOL ;
  input_76_7 : BOOL ;
  input_77_0 : BOOL ;
  input_77_1 : BOOL ;
  input_77_2 : BOOL ;
  input_77_3 : BOOL ;
  input_77_4 : BOOL ;
  input_77_5 : BOOL ;
  input_77_6 : BOOL ;
  input_77_7 : BOOL ;
  input_78_0 : BOOL ;
  input_78_1 : BOOL ;
  input_78_2 : BOOL ;
  input_78_3 : BOOL ;
  input_78_4 : BOOL ;
  input_78_5 : BOOL ;
  input_78_6 : BOOL ;
  input_78_7 : BOOL ;
  input_79_0 : BOOL ;
  input_79_1 : BOOL ;
  input_79_2 : BOOL ;
  input_79_3 : BOOL ;
  input_79_4 : BOOL ;
  input_79_5 : BOOL ;
  input_79_6 : BOOL ;
  input_79_7 : BOOL ;
  input_80_0 : BOOL ;
  input_80_1 : BOOL ;
  input_80_2 : BOOL ;
  input_80_3 : BOOL ;
  input_80_4 : BOOL ;
  input_80_5 : BOOL ;
  input_80_6 : BOOL ;
  input_80_7 : BOOL ;
  input_81_0 : BOOL ;
  input_81_1 : BOOL ;
  input_81_2 : BOOL ;
  input_81_3 : BOOL ;
  input_81_4 : BOOL ;
  input_81_5 : BOOL ;
  input_81_6 : BOOL ;
  input_81_7 : BOOL ;
  input_82_0 : BOOL ;
  input_82_1 : BOOL ;
  input_82_2 : BOOL ;
  input_82_3 : BOOL ;
  input_82_4 : BOOL ;
  input_82_5 : BOOL ;
  input_82_6 : BOOL ;
  input_82_7 : BOOL ;
  input_83_0 : BOOL ;
  input_83_1 : BOOL ;
  input_83_2 : BOOL ;
  input_83_3 : BOOL ;
  input_83_4 : BOOL ;
  input_83_5 : BOOL ;
  input_83_6 : BOOL ;
  input_83_7 : BOOL ;
  input_84_0 : BOOL ;
  input_84_1 : BOOL ;
  input_84_2 : BOOL ;
  input_84_3 : BOOL ;
  input_84_4 : BOOL ;
  input_84_5 : BOOL ;
  input_84_6 : BOOL ;
  input_84_7 : BOOL ;
  input_85_0 : BOOL ;
  input_85_1 : BOOL ;
  input_85_2 : BOOL ;
  input_85_3 : BOOL ;
  input_85_4 : BOOL ;
  input_85_5 : BOOL ;
  input_85_6 : BOOL ;
  input_85_7 : BOOL ;
  input_86_0 : BOOL ;
  input_86_1 : BOOL ;
  input_86_2 : BOOL ;
  input_86_3 : BOOL ;
  input_86_4 : BOOL ;
  input_86_5 : BOOL ;
  input_86_6 : BOOL ;
  input_86_7 : BOOL ;
  input_87_0 : BOOL ;
  input_87_1 : BOOL ;
  input_87_2 : BOOL ;
  input_87_3 : BOOL ;
  input_87_4 : BOOL ;
  input_87_5 : BOOL ;
  input_87_6 : BOOL ;
  input_87_7 : BOOL ;
  input_88_0 : BOOL ;
  input_88_1 : BOOL ;
  input_88_2 : BOOL ;
  input_88_3 : BOOL ;
  input_88_4 : BOOL ;
  input_88_5 : BOOL ;
  input_88_6 : BOOL ;
  input_88_7 : BOOL ;
  input_89_0 : BOOL ;
  input_89_1 : BOOL ;
  input_89_2 : BOOL ;
  input_89_3 : BOOL ;
  input_89_4 : BOOL ;
  input_89_5 : BOOL ;
  input_89_6 : BOOL ;
  input_89_7 : BOOL ;
  input_90_0 : BOOL ;
  input_90_1 : BOOL ;
  input_90_2 : BOOL ;
  input_90_3 : BOOL ;
  input_90_4 : BOOL ;
  input_90_5 : BOOL ;
  input_90_6 : BOOL ;
  input_90_7 : BOOL ;
  input_91_0 : BOOL ;
  input_91_1 : BOOL ;
  input_91_2 : BOOL ;
  input_91_3 : BOOL ;
  input_91_4 : BOOL ;
  input_91_5 : BOOL ;
  input_91_6 : BOOL ;
  input_91_7 : BOOL ;
  input_92_0 : BOOL ;
  input_92_1 : BOOL ;
  input_92_2 : BOOL ;
  input_92_3 : BOOL ;
  input_92_4 : BOOL ;
  input_92_5 : BOOL ;
  input_92_6 : BOOL ;
  input_92_7 : BOOL ;
  input_93_0 : BOOL ;
  input_93_1 : BOOL ;
  input_93_2 : BOOL ;
  input_93_3 : BOOL ;
  input_93_4 : BOOL ;
  input_93_5 : BOOL ;
  input_93_6 : BOOL ;
  input_93_7 : BOOL ;
  input_94_0 : BOOL ;
  input_94_1 : BOOL ;
  input_94_2 : BOOL ;
  input_94_3 : BOOL ;
  input_94_4 : BOOL ;
  input_94_5 : BOOL ;
  input_94_6 : BOOL ;
  input_94_7 : BOOL ;
  input_95_0 : BOOL ;
  input_95_1 : BOOL ;
  input_95_2 : BOOL ;
  input_95_3 : BOOL ;
  input_95_4 : BOOL ;
  input_95_5 : BOOL ;
  input_95_6 : BOOL ;
  input_95_7 : BOOL ;
  input_96_0 : BOOL ;
  input_96_1 : BOOL ;
  input_96_2 : BOOL ;
  input_96_3 : BOOL ;
  input_96_4 : BOOL ;
  input_96_5 : BOOL ;
  input_96_6 : BOOL ;
  input_96_7 : BOOL ;
  input_97_0 : BOOL ;
  input_97_1 : BOOL ;
  input_97_2 : BOOL ;
  input_97_3 : BOOL ;
  input_97_4 : BOOL ;
  input_97_5 : BOOL ;
  input_97_6 : BOOL ;
  input_97_7 : BOOL ;
  input_98_0 : BOOL ;
  input_98_1 : BOOL ;
  input_98_2 : BOOL ;
  input_98_3 : BOOL ;
  input_98_4 : BOOL ;
  input_98_5 : BOOL ;
  input_98_6 : BOOL ;
  input_98_7 : BOOL ;
  input_99_0 : BOOL ;
  input_99_1 : BOOL ;
  input_99_2 : BOOL ;
  input_99_3 : BOOL ;
  input_99_4 : BOOL ;
  input_99_5 : BOOL ;
  input_99_6 : BOOL ;
  input_99_7 : BOOL ;
  input_100_0 : BOOL ;
  input_100_1 : BOOL ;
  input_100_2 : BOOL ;
  input_100_3 : BOOL ;
  input_100_4 : BOOL ;
  input_100_5 : BOOL ;
  input_100_6 : BOOL ;
  input_100_7 : BOOL ;
  input_101_0 : BOOL ;
  input_101_1 : BOOL ;
  input_101_2 : BOOL ;
  input_101_3 : BOOL ;
  input_101_4 : BOOL ;
  input_101_5 : BOOL ;
  input_101_6 : BOOL ;
  input_101_7 : BOOL ;
  input_102_0 : BOOL ;
  input_102_1 : BOOL ;
  input_102_2 : BOOL ;
  input_102_3 : BOOL ;
  input_102_4 : BOOL ;
  input_102_5 : BOOL ;
  input_102_6 : BOOL ;
  input_102_7 : BOOL ;
  input_103_0 : BOOL ;
  input_103_1 : BOOL ;
  input_103_2 : BOOL ;
  input_103_3 : BOOL ;
  input_103_4 : BOOL ;
  input_103_5 : BOOL ;
  input_103_6 : BOOL ;
  input_103_7 : BOOL ;
  input_104_0 : BOOL ;
  input_104_1 : BOOL ;
  input_104_2 : BOOL ;
  input_104_3 : BOOL ;
  input_104_4 : BOOL ;
  input_104_5 : BOOL ;
  input_104_6 : BOOL ;
  input_104_7 : BOOL ;
  input_105_0 : BOOL ;
  input_105_1 : BOOL ;
  input_105_2 : BOOL ;
  input_105_3 : BOOL ;
  input_105_4 : BOOL ;
  input_105_5 : BOOL ;
  input_105_6 : BOOL ;
  input_105_7 : BOOL ;
  input_106_0 : BOOL ;
  input_106_1 : BOOL ;
  input_106_2 : BOOL ;
  input_106_3 : BOOL ;
  input_106_4 : BOOL ;
  input_106_5 : BOOL ;
  input_106_6 : BOOL ;
  input_106_7 : BOOL ;
  input_107_0 : BOOL ;
  input_107_1 : BOOL ;
  input_107_2 : BOOL ;
  input_107_3 : BOOL ;
  input_107_4 : BOOL ;
  input_107_5 : BOOL ;
  input_107_6 : BOOL ;
  input_107_7 : BOOL ;
  input_108_0 : BOOL ;
  input_108_1 : BOOL ;
  input_108_2 : BOOL ;
  input_108_3 : BOOL ;
  input_108_4 : BOOL ;
  input_108_5 : BOOL ;
  input_108_6 : BOOL ;
  input_108_7 : BOOL ;
  input_109_0 : BOOL ;
  input_109_1 : BOOL ;
  input_109_2 : BOOL ;
  input_109_3 : BOOL ;
  input_109_4 : BOOL ;
  input_109_5 : BOOL ;
  input_109_6 : BOOL ;
  input_109_7 : BOOL ;
  input_110_0 : BOOL ;
  input_110_1 : BOOL ;
  input_110_2 : BOOL ;
  input_110_3 : BOOL ;
  input_110_4 : BOOL ;
  input_110_5 : BOOL ;
  input_110_6 : BOOL ;
  input_110_7 : BOOL ;
  input_111_0 : BOOL ;
  input_111_1 : BOOL ;
  input_111_2 : BOOL ;
  input_111_3 : BOOL ;
  input_111_4 : BOOL ;
  input_111_5 : BOOL ;
  input_111_6 : BOOL ;
  input_111_7 : BOOL ;
  input_112_0 : BOOL ;
  input_112_1 : BOOL ;
  input_112_2 : BOOL ;
  input_112_3 : BOOL ;
  input_112_4 : BOOL ;
  input_112_5 : BOOL ;
  input_112_6 : BOOL ;
  input_112_7 : BOOL ;
  input_113_0 : BOOL ;
  input_113_1 : BOOL ;
  input_113_2 : BOOL ;
  input_113_3 : BOOL ;
  input_113_4 : BOOL ;
  input_113_5 : BOOL ;
  input_113_6 : BOOL ;
  input_113_7 : BOOL ;
  input_114_0 : BOOL ;
  input_114_1 : BOOL ;
  input_114_2 : BOOL ;
  input_114_3 : BOOL ;
  input_114_4 : BOOL ;
  input_114_5 : BOOL ;
  input_114_6 : BOOL ;
  input_114_7 : BOOL ;
  input_115_0 : BOOL ;
  input_115_1 : BOOL ;
  input_115_2 : BOOL ;
  input_115_3 : BOOL ;
  input_115_4 : BOOL ;
  input_115_5 : BOOL ;
  input_115_6 : BOOL ;
  input_115_7 : BOOL ;
  input_116_0 : BOOL ;
  input_116_1 : BOOL ;
  input_116_2 : BOOL ;
  input_116_3 : BOOL ;
  input_116_4 : BOOL ;
  input_116_5 : BOOL ;
  input_116_6 : BOOL ;
  input_116_7 : BOOL ;
  input_117_0 : BOOL ;
  input_117_1 : BOOL ;
  input_117_2 : BOOL ;
  input_117_3 : BOOL ;
  input_117_4 : BOOL ;
  input_117_5 : BOOL ;
  input_117_6 : BOOL ;
  input_117_7 : BOOL ;
  input_118_0 : BOOL ;
  input_118_1 : BOOL ;
  input_118_2 : BOOL ;
  input_118_3 : BOOL ;
  input_118_4 : BOOL ;
  input_118_5 : BOOL ;
  input_118_6 : BOOL ;
  input_118_7 : BOOL ;
  input_119_0 : BOOL ;
  input_119_1 : BOOL ;
  input_119_2 : BOOL ;
  input_119_3 : BOOL ;
  input_119_4 : BOOL ;
  input_119_5 : BOOL ;
  input_119_6 : BOOL ;
  input_119_7 : BOOL ;
  input_120_0 : BOOL ;
  input_120_1 : BOOL ;
  input_120_2 : BOOL ;
  input_120_3 : BOOL ;
  input_120_4 : BOOL ;
  input_120_5 : BOOL ;
  input_120_6 : BOOL ;
  input_120_7 : BOOL ;
  input_121_0 : BOOL ;
  input_121_1 : BOOL ;
  input_121_2 : BOOL ;
  input_121_3 : BOOL ;
  input_121_4 : BOOL ;
  input_121_5 : BOOL ;
  input_121_6 : BOOL ;
  input_121_7 : BOOL ;
  input_122_0 : BOOL ;
  input_122_1 : BOOL ;
  input_122_2 : BOOL ;
  input_122_3 : BOOL ;
  input_122_4 : BOOL ;
  input_122_5 : BOOL ;
  input_122_6 : BOOL ;
  input_122_7 : BOOL ;
  input_123_0 : BOOL ;
  input_123_1 : BOOL ;
  input_123_2 : BOOL ;
  input_123_3 : BOOL ;
  input_123_4 : BOOL ;
  input_123_5 : BOOL ;
  input_123_6 : BOOL ;
  input_123_7 : BOOL ;
  input_124_0 : BOOL ;
  input_124_1 : BOOL ;
  input_124_2 : BOOL ;
  input_124_3 : BOOL ;
  input_124_4 : BOOL ;
  input_124_5 : BOOL ;
  input_124_6 : BOOL ;
  input_124_7 : BOOL ;
  input_125_0 : BOOL ;
  input_125_1 : BOOL ;
  input_125_2 : BOOL ;
  input_125_3 : BOOL ;
  input_125_4 : BOOL ;
  input_125_5 : BOOL ;
  input_125_6 : BOOL ;
  input_125_7 : BOOL ;
  input_126_0 : BOOL ;
  input_126_1 : BOOL ;
  input_126_2 : BOOL ;
  input_126_3 : BOOL ;
  input_126_4 : BOOL ;
  input_126_5 : BOOL ;
  input_126_6 : BOOL ;
  input_126_7 : BOOL ;
  input_127_0 : BOOL ;
  input_127_1 : BOOL ;
  input_127_2 : BOOL ;
  input_127_3 : BOOL ;
  input_127_4 : BOOL ;
  input_127_5 : BOOL ;
  input_127_6 : BOOL ;
  input_127_7 : BOOL ;
  input_128_0 : BOOL ;
  input_128_1 : BOOL ;
  input_128_2 : BOOL ;
  input_128_3 : BOOL ;
  input_128_4 : BOOL ;
  input_128_5 : BOOL ;
  input_128_6 : BOOL ;
  input_128_7 : BOOL ;
  input_129_0 : BOOL ;
  input_129_1 : BOOL ;
  input_129_2 : BOOL ;
  input_129_3 : BOOL ;
  input_129_4 : BOOL ;
  input_129_5 : BOOL ;
  input_129_6 : BOOL ;
  input_129_7 : BOOL ;
  reserve : ARRAY  [130 .. 1000 ] OF BYTE ;
END_VAR
BEGIN
NETWORK
TITLE = UR1
//!!!!! Beispiel !!!!!  
//
      L     IW 4;
      T     DIW 4;
      L     IW 8;
      T     DIW 8;
      L     IW 12;
      T     DIW 12;
      L     IW 16;
      T     DIW 16;
      L     IW 20;
      T     DIW 20;
      L     IW 24;
      T     DIW 24;
//      L     IW    28
//      T     DIW   28
//      L     IW    32
//      T     DIW   32
//      L     ID    36
//      T     DID   36
//      L     ID    40
//      T     DID   40
//      L     IW    44
//      T     DIW   44
//      L     IW    48
//      T     DIW   48
//      L     IW    52
//      T     DIW   52
NETWORK
TITLE = ET200B Module
//!!!!! Beispiel !!!!!  
//
//      L     ID    56
//      T     DID   56
//      L     ID    60
//      T     DID   60
//      L     ID    64
//      T     DID   64
//     L     ID    68
//     T     DID   68
//      L     ID    70
//      T     DID   70
//      L     ID    74
//      T     DID   74
//      L     ID    78
//      T     DID   78
//      L     ID    80
//      T     DID   80
//      L     ID    84
//      T     DID   84
//      L     ID    88
//      T     DID   88
//      L     ID    90
//      T     DID   90
//      L     ID    94
//      T     DID   94
//      L     ID    98
//      T     DID   98
//      L     ID   100
//      T     DID  100
//      L     ID   104
//      T     DID  104
END_FUNCTION_BLOCK

